# B&R Automation Studio project Nitto (part 17)

#### ac_loadRecipeMain.st
```iecst
(********************************************************************
 * COPYRIGHT -- Microsoft
 ********************************************************************
 * Programm: MAIN
 * Datei: ac_loadRecipeMain.st
 * Autor: awalz
 * Erstellt: 29. Juli 2014
 ********************************************************************
 * Implementierung des Programms MAIN
 ********************************************************************)

(* Fügt eine neue Aktion zum IEC Programm oder Bibliothek *)
ACTION ac_loadRecipeMain:

		// cutting units
		memcpy(ADR(machine.cuttingunit1.data.recipe),ADR(gApplRecipe.cutUnit1),SIZEOF(machine.cuttingunit1.data.recipe));
		memcpy(ADR(machine.cuttingunit2.data.recipe),ADR(gApplRecipe.cutUnit2),SIZEOF(machine.cuttingunit2.data.recipe));
		memcpy(ADR(machine.cuttingunit1.data.general),ADR(gApplRecipe.general),SIZEOF(machine.cuttingunit1.data.general));
		memcpy(ADR(machine.cuttingunit2.data.general),ADR(gApplRecipe.general),SIZEOF(machine.cuttingunit2.data.general));
		memcpy(ADR(machine.cuttingunit1.data.machdata),ADR(gMachRecipe.cut1),SIZEOF(machine.cuttingunit1.data.machdata));
		memcpy(ADR(machine.cuttingunit2.data.machdata),ADR(gMachRecipe.cut2),SIZEOF(machine.cuttingunit2.data.machdata));
//		machine.cuttingunit2.ctrl.getNextCuttPos.setCutOffset.UpdateRecipe := TRUE;
//		machine.cuttingunit2.ctrl.getNextCuttPos.setCutOffset.setvalueVisuRecipe := gApplRecipe.cutUnit2.RmOffset;
	(*	machine.cuttingunit1.data.machdata.position := 1000000;*)
		machine.cuttingunit1.data.general.periodLength := gApplRecipe.general.periodLength;
		machine.cuttingunit1.data.recipe.tool.gearRatioMotor := 5;(* weil die mit 0 überschrieben werden da der Krebs wieder Misst gebaut hat*)
		machine.cuttingunit1.data.recipe.tool.cogmodul :=3175.0;
		machine.cuttingunit1.data.newRecipe := TRUE;
		machine.cuttingunit2.data.recipe.tool.gearRatioMotor := 5;
		machine.cuttingunit2.data.recipe.tool.cogmodul :=3175.0;
	(*	machine.cuttingunit2.data.machdata.position := 3400000;*)
		machine.cuttingunit2.data.general.periodLength := gApplRecipe.general.periodLength;
		machine.cuttingunit2.markpoints.RegMarkPosition := -540000;
		machine.cuttingunit2.data.machdata.position := 850000;
		machine.cuttingunit2.data.newRecipe := TRUE;
//		machine.cuttingunit2.markpoints.RegMarkPosition := -540000; //Abstand vom Sensor zu Stanzmitte

		machine.masterModul.data.lenght1 := gApplRecipe.general.lenght1;
		machine.masterModul.data.lenght1 := gApplRecipe.general.lenght1;

		// master // general
		machine.masterModul.data.maxSpeed := gApplRecipe.general.maxVelocity;
		machine.masterModul.data.periodLength := gApplRecipe.general.periodLength;
		machine.masterModul.data.startSpeed := gApplRecipe.general.startVelocity;
		machine.masterModul.data.lenght1 := gApplRecipe.general.lenght1;
		machine.masterModul.data.lenght2 := gApplRecipe.general.lenght2;
		machine.masterModul.data.speedToCycleWebturrit := gApplRecipe.general.speedToCycleWebturrit;

		// unwinder drive side
		machine.UnwinderUnit.unwinderDrv.data.recipeData.maxDiamTension := gApplRecipe.UnwinderDrvSide.maxDiamTension;
		machine.UnwinderUnit.unwinderDrv.data.recipeData.minDiamTension := gApplRecipe.UnwinderDrvSide.minDiamTension;
		machine.UnwinderUnit.unwinderDrv.data.recipeData.mode := gApplRecipe.UnwinderDrvSide.mode;
		machine.UnwinderUnit.unwinderDrv.data.recipeData.reverse := gApplRecipe.UnwinderDrvSide.reverse;
		machine.UnwinderUnit.unwinderDrv.data.recipeData.warnDiam := gApplRecipe.UnwinderDrvSide.warnDiam;
		machine.UnwinderUnit.unwinderDrv.data.recipeData.stopDiam := gApplRecipe.UnwinderDrvSide.stopDiam;
		machine.UnwinderUnit.unwinderDrv.data.machData.axistyp := 1;	(*(-1: winder, +1: unwinder).*)
		// unwinder op side
		machine.UnwinderUnit.unwinderOp.data.recipeData.maxDiamTension := gApplRecipe.UnwinderOpSide.maxDiamTension;
		machine.UnwinderUnit.unwinderOp.data.recipeData.minDiamTension := gApplRecipe.UnwinderOpSide.minDiamTension;
		machine.UnwinderUnit.unwinderOp.data.recipeData.mode := gApplRecipe.UnwinderOpSide.mode;
		machine.UnwinderUnit.unwinderOp.data.recipeData.reverse := gApplRecipe.UnwinderOpSide.reverse;
		machine.UnwinderUnit.unwinderOp.data.recipeData.warnDiam := gApplRecipe.UnwinderOpSide.warnDiam;
		machine.UnwinderUnit.unwinderOp.data.recipeData.stopDiam := gApplRecipe.UnwinderOpSide.stopDiam;
		machine.UnwinderUnit.unwinderOp.data.machData.axistyp := 1;(*(-1: winder, +1: unwinder).*)
		// grid winder left
		machine.turngridwinder.gridwinderleft.data.recipeData.maxDiamTension := gApplRecipe.gridwinderleft.maxDiamTension;
		machine.turngridwinder.gridwinderleft.data.recipeData.minDiamTension := gApplRecipe.gridwinderleft.minDiamTension;
		machine.turngridwinder.gridwinderleft.data.recipeData.mode := gApplRecipe.gridwinderleft.mode;
		machine.turngridwinder.gridwinderleft.data.recipeData.reverse := gApplRecipe.gridwinderleft.reverse;
		machine.turngridwinder.gridwinderleft.data.recipeData.warnDiam := gApplRecipe.gridwinderleft.warnDiam;
		machine.turngridwinder.gridwinderleft.data.recipeData.stopDiam := gApplRecipe.gridwinderleft.stopDiam;
		machine.turngridwinder.gridwinderleft.data.machData.axistyp := - 1;(*(-1: winder, +1: unwinder).*)

		// grid winder right
		machine.turngridwinder.gridwinderright.data.recipeData.maxDiamTension := gApplRecipe.gridwinderright.maxDiamTension;
		machine.turngridwinder.gridwinderright.data.recipeData.minDiamTension := gApplRecipe.gridwinderright.minDiamTension;
		machine.turngridwinder.gridwinderright.data.recipeData.mode := gApplRecipe.gridwinderright.mode;
		machine.turngridwinder.gridwinderright.data.recipeData.reverse := gApplRecipe.gridwinderright.reverse;
		machine.turngridwinder.gridwinderright.data.recipeData.warnDiam := gApplRecipe.gridwinderright.warnDiam;
		machine.turngridwinder.gridwinderright.data.recipeData.stopDiam := gApplRecipe.gridwinderright.stopDiam;
		machine.turngridwinder.gridwinderright.data.machData.axistyp := - 1;
		// catch belt
		machine.catchbelt.ctrl.mode := gApplRecipe.catchbelt.mode;
		machine.catchbelt.axis.setGearRatio.enable := gApplRecipe.catchbelt.offsetOnOff;
		machine.catchbelt.axis.setGearRatio.UpdateRecipe := TRUE;
		machine.catchbelt.axis.setGearRatio.setvalueVisuRecipe := gApplRecipe.catchbelt.setvaluevisu;

		// conveyor
		machine.conveyor.ctrl.mode := gApplRecipe.conveyor.mode;
		machine.conveyor.axis.setGearRatio.enable := gApplRecipe.conveyor.offsetOnOff;
		machine.conveyor.axis.setGearRatio.UpdateRecipe := TRUE;
		machine.conveyor.axis.setGearRatio.setvalueVisuRecipe := gApplRecipe.conveyor.setvaluevisu;
		machine.conveyor.counters.setPieces := gApplRecipe.conveyor.setPieces;
		machine.conveyor.counters.validpieces := gApplRecipe.conveyor.validPieces;
		// long cuttter
		machine.longcutter.ctrl.mode := gApplRecipe.longcutter.mode;
		machine.longcutter.axis.setGearRatio.enable := gApplRecipe.longcutter.offsetOnOff;
		machine.longcutter.axis.setGearRatio.UpdateRecipe := TRUE;
		machine.longcutter.axis.setGearRatio.setvalueVisuRecipe := gApplRecipe.longcutter.setvaluevisu;

		// pull break station (pull belt)
		machine.pullbreakSt.axis.setGearRatio.enable := gApplRecipe.pullbelt.offsetOnOff;
		machine.pullbreakSt.axis.setGearRatio.UpdateRecipe := TRUE;
		machine.pullbreakSt.axis.setGearRatio.setvalueVisuRecipe := gApplRecipe.pullbelt.setvaluevisu;

		// Webbuffer
		machine.webbuffer.data.recipe.mode := gApplRecipe.tensionMeas.mode;
		machine.webbuffer.data.recipe.SetTension := gApplRecipe.tensionMeas.webTension;
END_ACTION
```

#### ac_loadMach_toRecipeMain.st
```iecst
(********************************************************************
 * COPYRIGHT -- Microsoft
 ********************************************************************
 * Programm: MAIN
 * Datei: ac_loadMach_toRecipeMain.st
 * Autor: awalz
 * Erstellt: 29. Juli 2014
 ********************************************************************
 * Implementierung des Programms MAIN
 ********************************************************************)

(* Fügt eine neue Aktion zum IEC Programm oder Bibliothek *)
ACTION ac_loadMach_toRecipeMain:

		// 2012-12-19 /schoenefeldr/
		// Copy recipe data from application recipe (actually active in the machine) into the selected recipe
		memcpy(ADR(RecipeEdit.cutUnit1),ADR(machine.cuttingunit1.data.recipe),SIZEOF(RecipeEdit.cutUnit1));
		memcpy(ADR(RecipeEdit.cutUnit2),ADR(machine.cuttingunit2.data.recipe),SIZEOF(RecipeEdit.cutUnit2));

//		RecipeEdit.cutUnit1.RmOffset := machine.cuttingunit1.ctrl.getNextCuttPos.setCutOffset.setvalueVisu;	 // OKrebs 15.09.14 //Damit der richtige Offsetwert in die perm Daten geschrieben wird
//		RecipeEdit.cutUnit2.RmOffset := machine.cuttingunit2.ctrl.getNextCuttPos.setCutOffset.setvalueVisu;  // OKrebs 15.09.14 //Damit der richtige Offsetwert in die perm Daten geschrieben wird
		RecipeEdit.general.lenght1 := machine.masterModul.data.lenght1; // OKrebs 17.09.14
		RecipeEdit.general.lenght2 := machine.masterModul.data.lenght2; // OKrebs 17.09.14
		RecipeEdit.general.speedToCycleWebturrit := machine.masterModul.data.speedToCycleWebturrit;

		machine.cuttingunit1.data.recipe.tool.gearRatioMotor := 5;(* weil die mit 0 überschrieben werden da der Krebs wieder Misst gebaut hat*)
		machine.cuttingunit1.data.recipe.tool.cogmodul :=3175.0;
		machine.cuttingunit2.data.recipe.tool.gearRatioMotor := 5;
		machine.cuttingunit2.data.recipe.tool.cogmodul :=3175.0;
		machine.cuttingunit2.markpoints.RegMarkPosition := -540000;
		machine.cuttingunit2.data.machdata.position := 850000;
		machine.cuttingunit2.data.general.periodLength := gApplRecipe.general.periodLength; //460000;
		(*machine.cuttingunit2.data.recipe.RmOffset*); (* muss noch irgendwie zu ende gebracht werden*)

		// unwinder drive side
		RecipeEdit.UnwinderDrvSide.maxDiamTension := machine.UnwinderUnit.unwinderDrv.data.recipeData.maxDiamTension;
		RecipeEdit.UnwinderDrvSide.minDiamTension := machine.UnwinderUnit.unwinderDrv.data.recipeData.minDiamTension;
		RecipeEdit.UnwinderDrvSide.mode := machine.UnwinderUnit.unwinderDrv.data.recipeData.mode;
		RecipeEdit.UnwinderDrvSide.reverse := machine.UnwinderUnit.unwinderDrv.data.recipeData.reverse;
		RecipeEdit.UnwinderDrvSide.warnDiam := machine.UnwinderUnit.unwinderDrv.data.recipeData.warnDiam;
		RecipeEdit.UnwinderDrvSide.stopDiam := machine.UnwinderUnit.unwinderDrv.data.recipeData.stopDiam;
//		RecipeEdit.UnwinderDrvSide.data.machData.GEAR_RATIO := 8;(*gMachRecipe.UnwinderDrvSide.GEAR_RATIO;*)
//		RecipeEdit.UnwinderDrvSide.machData.axistyp := 1;	(*(-1: winder, +1: unwinder).*)
		// unwinder op side
		RecipeEdit.UnwinderOpSide.maxDiamTension := machine.UnwinderUnit.unwinderOp.data.recipeData.maxDiamTension;
		RecipeEdit.UnwinderOpSide.minDiamTension := machine.UnwinderUnit.unwinderOp.data.recipeData.minDiamTension;
		RecipeEdit.UnwinderOpSide.mode := machine.UnwinderUnit.unwinderOp.data.recipeData.mode;
		RecipeEdit.UnwinderOpSide.reverse := machine.UnwinderUnit.unwinderOp.data.recipeData.reverse;
		RecipeEdit.UnwinderOpSide.warnDiam := machine.UnwinderUnit.unwinderOp.data.recipeData.warnDiam;
		RecipeEdit.UnwinderOpSide.stopDiam := machine.UnwinderUnit.unwinderOp.data.recipeData.stopDiam;
//		RecipeEdit.unwinderOp.data.machData.GEAR_RATIO := 8; (*gMachRecipe.UnwinderOpSide.GEAR_RATIO;*)
//		RecipeEdit.unwinderOp.data.machData.axistyp := 1;(*(-1: winder, +1: unwinder).*)
		// grid winder left
		RecipeEdit.gridwinderleft.maxDiamTension := machine.turngridwinder.gridwinderleft.data.recipeData.maxDiamTension;
		RecipeEdit.gridwinderleft.minDiamTension := machine.turngridwinder.gridwinderleft.data.recipeData.minDiamTension;
		RecipeEdit.gridwinderleft.mode := machine.turngridwinder.gridwinderleft.data.recipeData.mode;
		RecipeEdit.gridwinderleft.reverse := machine.turngridwinder.gridwinderleft.data.recipeData.reverse;
		RecipeEdit.gridwinderleft.warnDiam := machine.turngridwinder.gridwinderleft.data.recipeData.warnDiam;
		RecipeEdit.gridwinderleft.stopDiam := machine.turngridwinder.gridwinderleft.data.recipeData.stopDiam;
//		RecipeEdit.gridwinderleft.data.machData.GEAR_RATIO := 3; (*gMachRecipe.gridwinderleft.GEAR_RATIO;*)
//		RecipeEdit.gridwinderleft.data.machData.axistyp := - 1;(*(-1: winder, +1: unwinder).*)
		// grid winder right
		RecipeEdit.gridwinderright.maxDiamTension := machine.turngridwinder.gridwinderright.data.recipeData.maxDiamTension;
		RecipeEdit.gridwinderright.minDiamTension := machine.turngridwinder.gridwinderright.data.recipeData.minDiamTension;
		RecipeEdit.gridwinderright.mode := machine.turngridwinder.gridwinderright.data.recipeData.mode;
		RecipeEdit.gridwinderright.reverse := machine.turngridwinder.gridwinderright.data.recipeData.reverse;
		RecipeEdit.gridwinderright.warnDiam := machine.turngridwinder.gridwinderright.data.recipeData.warnDiam;
		RecipeEdit.gridwinderright.stopDiam := machine.turngridwinder.gridwinderright.data.recipeData.stopDiam;
//		RecipeEdit.gridwinderright.data.machData.GEAR_RATIO := 3; (*gMachRecipe.gridwinderleft.GEAR_RATIO;*)
//		RecipeEdit.gridwinderright.data.machData.axistyp := - 1;(*(-1: winder, +1: unwinder).*)
		// catch belt
		RecipeEdit.catchbelt.mode := machine.catchbelt.ctrl.mode;
		RecipeEdit.catchbelt.offsetOnOff := machine.catchbelt.axis.setGearRatio.enable;
		RecipeEdit.catchbelt.setvaluevisu := machine.catchbelt.axis.setGearRatio.setvalueVisu;

		// conveyor
		RecipeEdit.conveyor.mode := machine.conveyor.ctrl.mode;
		RecipeEdit.conveyor.offsetOnOff := machine.conveyor.axis.setGearRatio.enable;
		RecipeEdit.conveyor.setvaluevisu := machine.conveyor.axis.setGearRatio.setvalueVisu;

		// long cuttter
		RecipeEdit.longcutter.mode := machine.longcutter.ctrl.mode;
		RecipeEdit.longcutter.offsetOnOff := machine.longcutter.axis.setGearRatio.enable;
		RecipeEdit.longcutter.setvaluevisu := machine.longcutter.axis.setGearRatio.setvalueVisu;

		// pull break station (pull belt)
		RecipeEdit.pullbelt.offsetOnOff := machine.pullbreakSt.axis.setGearRatio.enable;
		RecipeEdit.pullbelt.setvaluevisu := machine.pullbreakSt.axis.setGearRatio.setvalueVisu;

		// Webbuffer Tension
		RecipeEdit.tensionMeas.mode := machine.webbuffer.data.recipe.mode;
		RecipeEdit.tensionMeas.webTension := machine.webbuffer.data.recipe.SetTension;
		/////////////////////////////////////////////////////////////////////////////////////////////////////////////////////////////

END_ACTION
```

#### ac_saveMachData.st
```iecst
(********************************************************************
 * COPYRIGHT -- Microsoft
 ********************************************************************
 * Programm: MAIN
 * Datei: ac_saveMachData.st
 * Autor: okrebs
 * Erstellt: 30. Juli 2014
 ********************************************************************
 * Implementierung des Programms MAIN
 ********************************************************************)

(* speichern der Maschinendaten zu MAIN_Variablen *)
ACTION ac_saveMachData:

		// distances
		machine.cuttingunit2.data.machdata.position := 850000;
		machine.cuttingunit1.data.recipe.tool.gearRatioMotor := 5;(* weil die mit 0 überschrieben werden da der Krebs wieder Misst gebaut hat*)
		machine.cuttingunit1.data.recipe.tool.cogmodul :=3175.0;
		machine.cuttingunit2.data.recipe.tool.gearRatioMotor := 5;
		machine.cuttingunit2.data.recipe.tool.cogmodul :=3175.0;
		machine.cuttingunit2.markpoints.RegMarkPosition := -540000;
	(*	machine.cuttingunit2.data.machdata.position := 540000;*)

		// unwinder drive side
		machine.UnwinderUnit.unwinderDrv.data.machData.coreDiam := gMachRecipe.UnwinderDrvSide.coreDiam;
		machine.UnwinderUnit.unwinderDrv.data.machData.frictionCompensation := gMachRecipe.UnwinderDrvSide.frictionCompensation;
		machine.UnwinderUnit.unwinderDrv.data.machData.GEAR_RATIO := 8;(*gMachRecipe.UnwinderDrvSide.GEAR_RATIO;*)
		machine.UnwinderUnit.unwinderDrv.data.machData.velocityOverride := gMachRecipe.UnwinderDrvSide.velocityOverride;
		machine.UnwinderUnit.unwinderDrv.data.machData.axistyp := 1;	(*(-1: winder, +1: unwinder).*)
		// unwinder op side
		machine.UnwinderUnit.unwinderOp.data.machData.coreDiam := gMachRecipe.UnwinderOpSide.coreDiam;
		machine.UnwinderUnit.unwinderOp.data.machData.frictionCompensation := gMachRecipe.UnwinderOpSide.frictionCompensation;
		machine.UnwinderUnit.unwinderOp.data.machData.GEAR_RATIO := 8; (*gMachRecipe.UnwinderOpSide.GEAR_RATIO;*)
		machine.UnwinderUnit.unwinderOp.data.machData.velocityOverride := gMachRecipe.UnwinderOpSide.velocityOverride;
		machine.UnwinderUnit.unwinderOp.data.machData.axistyp := 1;(*(-1: winder, +1: unwinder).*)
		// grid winder left
		machine.turngridwinder.gridwinderleft.data.machData.coreDiam := gMachRecipe.gridwinderleft.coreDiam;
		machine.turngridwinder.gridwinderleft.data.machData.frictionCompensation := gMachRecipe.gridwinderleft.frictionCompensation;
		machine.turngridwinder.gridwinderleft.data.machData.GEAR_RATIO := 3; (*gMachRecipe.gridwinderleft.GEAR_RATIO;*)
		machine.turngridwinder.gridwinderleft.data.machData.velocityOverride := gMachRecipe.gridwinderleft.velocityOverride;
		machine.turngridwinder.gridwinderleft.data.machData.axistyp := - 1;(*(-1: winder, +1: unwinder).*)
		// grid winder right
		machine.turngridwinder.gridwinderright.data.machData.coreDiam := gMachRecipe.gridwinderright.coreDiam;
		machine.turngridwinder.gridwinderright.data.machData.frictionCompensation := gMachRecipe.gridwinderright.frictionCompensation;
		machine.turngridwinder.gridwinderright.data.machData.GEAR_RATIO := 3; (*gMachRecipe.gridwinderright.GEAR_RATIO;*)
		machine.turngridwinder.gridwinderright.data.machData.velocityOverride := gMachRecipe.gridwinderright.velocityOverride;
		machine.turngridwinder.gridwinderright.data.machData.axistyp := - 1;
		// pack belt
		machine.packbelt.data.acceleration	:= gMachRecipe.botTandemWind.WarnDiam;
		machine.packbelt.data.deceleration	:= gMachRecipe.botTandemWind.StopDiam;
		machine.packbelt.data.highSpeed		:= gMachRecipe.botTandemWind.MaxPressure;
		machine.packbelt.data.lowSpeed		:= gMachRecipe.botTandemWind.MinPressure;

END_ACTION
```

### Program Logical/MainMachineCtrl/dummy (IEC) - Programm

#### dummyCyclic.st - Zyklischer Code
```iecst
(********************************************************************
 * COPYRIGHT -- Microsoft
 ********************************************************************
 * Programm: dummy
 * Datei: dummyCyclic.st
 * Autor: awalz
 * Erstellt: 26. Juni 2014
 ********************************************************************
 * Implementierung des Programms dummy
 ********************************************************************)

PROGRAM _CYCLIC

(* TODO : Code hier einfügen *)

END_PROGRAM
```

#### dummyInit.st - Initialisierungscode
```iecst
(********************************************************************
 * COPYRIGHT -- Microsoft
 ********************************************************************
 * Programm: dummy
 * Datei: dummyInit.st
 * Autor: awalz
 * Erstellt: 26. Juni 2014
 ********************************************************************
 * Implementierung des Programms dummy
 ********************************************************************)

PROGRAM _INIT

(* TODO : Code hier einfügen *)
	gUnwinder := gUnwinder;
	gMaster1 := gMaster1; (*Virtueller Master*)
	gCut1 := gCut1; (*Stanzstation 1*)
	gCut2 := gCut2; (*Stanzstation 2*)
	gGridLeft := gGridLeft; (*Gitteraufwickler 1*)
	gGridRight := gGridRight; (*Gitteraufwickler 2*)
	gPBS1 := gPBS1; (*Zugstation 1*)
	gPBS2 := gPBS2; (*Zugstation 1*)
	gCatchBelt := gCatchBelt; (*Fangband*)
	gConvBelt := gConvBelt; (*Auslageband*)
	gUnwOp := gUnwOp; (*Abwickler Operatorseite*)
	gUnwDrv := gUnwDrv; (*Abwickler Antriebsseite*)
	gBuffer := gBuffer; (*Bahnspeicher*)
	gGridFeeder := gGridFeeder; (*Drehvorrichtung Gitterturm*)
	gLongCut := gLongCut; (*Drehvorrichtung Gitterturm*)
	gUnwFeeder := gUnwFeeder;
	gUnwFeeder_HW := gUnwFeeder_HW;
	gUnwFeeder_DrvIf := gUnwFeeder_DrvIf;
	gUnwFeeder_DiDoIf := gUnwFeeder_DiDoIf;
	gUnwFeeder_ModuleOk := gUnwFeeder_ModuleOk;
	// neu // OKrebs // 23.11.16
	gPackBelt := gPackBelt;
	gPackBelt_HW := gPackBelt_HW;
	gPackBelt_DrvIf := gPackBelt_DrvIf;
	gPackBelt_DiDoIf := gPackBelt_DiDoIf;
	gPackBelt_ModuleOk := gPackBelt_ModuleOk;
	// ende neu
END_PROGRAM
```

- Visualisation Logical/Visualization (not shown)

### Package Logical/pkgRecipe - recipe handling

### Program Logical/pkgRecipe/save2USB (IEC) - copy recipes from CF to USB

#### save2USB.st - Implementation code
```iecst
(********************************************************************
 * COPYRIGHT -- Bernecker + Rainer
 ********************************************************************
 * Program: USB_Test
 * File: USB_Test.st
 * Author: beutert
 * Created: February 10, 2012
 ********************************************************************
 * Implementation of program USB_Test
 ********************************************************************)

PROGRAM _INIT

LayerMessageBoxErrorUSB := INVISIBLE;
LayerMessageBoxCopyOkUSB := INVISIBLE;
strcpy(ADR(szRecipeDirName), ADR('Recipes'));
strcpy(ADR(szToolDirName), ADR('Tools'));

strcpy(ADR(szDirName), ADR(szRecipeDirName));

END_PROGRAM

PROGRAM _CYCLIC

IF (BackupRecipes2USB = TRUE) THEN
	BackupRecipes2USB := FALSE;
	strcpy(ADR(szDirName), ADR(szRecipeDirName));
	StartBackup2USB := TRUE;
END_IF;
IF (BackupTools2USB = TRUE) THEN
	BackupTools2USB := FALSE;
	strcpy(ADR(szDirName), ADR(szToolDirName));
	StartBackup2USB := TRUE;
END_IF;

CASE bStep OF
	ST_WAIT:
		IF (StartBackup2USB = TRUE) THEN
			bStep := CREATE_NODE_ID_LIST;
		END_IF;

	CREATE_NODE_ID_LIST:
		bStepOld := bStep;
		UsbNodeListGet_0.enable 									:= 1;
		UsbNodeListGet_0.pBuffer 									:= ADR(lNodeIdBuffer);
		UsbNodeListGet_0.bufferSize 							:= SIZEOF(lNodeIdBuffer);
		UsbNodeListGet_0.filterInterfaceClass 		:= asusb_CLASS_MASS_STORAGE;  (*set filter on mass storage devices*)
		UsbNodeListGet_0.filterInterfaceSubClass 	:= 0;	(*no filter is set *)
		UsbNodeListGet_0();

		wStatus := UsbNodeListGet_0.status;
		IF (wStatus = 0) THEN
    	bStep := READ_DEVICE_DATA;
		ELSIF UsbNodeListGet_0.status = ERR_FUB_BUSY THEN
			(* call FUB again *)
		ELSE
			bStep := ERROR_STEP;
		END_IF;

	READ_DEVICE_DATA:
		bStepOld := bStep;
		UsbNodeGet_0.enable 		:= 1;
		UsbNodeGet_0.nodeId 		:= lNodeIdBuffer[bNode];  				(*specific node is read out of node_id_buffer*)
		UsbNodeGet_0.pBuffer 		:= ADR(UsbDataBuffer[bNode]);  		(*data of specific node get stored in usb_data_buffer*)
		UsbNodeGet_0.bufferSize := SIZEOF(UsbDataBuffer[bNode]);  (*size of specific node is read out usb_data_buffer*)
		UsbNodeGet_0();

		wStatus := UsbNodeGet_0.status;

		IF (wStatus = 0) THEN
			bNode := bNode + 1;  (*next node to be read out of buffer*)
			IF (bNode = UsbNodeListGet_0.listNodes) THEN  (*last existing node is reached*)
				bNode := 0;
				bStep := GET_DESCRIPTOR;  (*all nodes are read out of buffer*)
			END_IF;
		ELSIF (wStatus = ERR_FUB_BUSY) THEN
			(* call FUB again *)
		ELSE
			bStep := ERROR_STEP;
		END_IF;

	GET_DESCRIPTOR:
		bStepOld := bStep;
		UsbDescriptorGet_0.enable 				:= 1;
		UsbDescriptorGet_0.nodeId 				:= lNodeIdBuffer[bNode];  (*specific node is read out of node_id_buffer*)
		UsbDescriptorGet_0.requestType 		:= 0;  (*Request for device*)
    UsbDescriptorGet_0.descriptorType := 1;  (*Determines the device descriptor*)
		UsbDescriptorGet_0.languageId 		:= 0;  (*for device and configuration descriptors*)
		UsbDescriptorGet_0.pBuffer 				:= ADR(DeviceDescriptor[bNode]);  (*descriptor-data of specific node get stored in device_descriptor-buffer*)
		UsbDescriptorGet_0.bufferSize 		:= SIZEOF(DeviceDescriptor[bNode]);  (*size of specific node is read out device_descriptor-buffer*)
		UsbDescriptorGet_0();

		wStatus := UsbDescriptorGet_0.status;

		IF (wStatus = 0) THEN
			bNode := bNode + 1;  (*next node to be read out of buffer*)
			IF (bNode = UsbNodeListGet_0.listNodes) THEN  (*last existing node is reached*)
				bNode := 0;
				bStep := CREATE_FILE_DEVICE;  (*all nodes are read out of buffer*)
			END_IF;
		ELSIF (wStatus = ERR_FUB_BUSY) THEN
			(* call FUB again *)
		ELSE
			bStep := ERROR_STEP;
		END_IF;

	CREATE_FILE_DEVICE:
		bStepOld := bStep;
		strcpy(ADR(szDeviceName), ADR('USBSTICK'));  (*fixed Device-Name get copied to device_name-Variable*)

		strcpy(ADR(szDeviceParam), ADR('/DEVICE='));  (*first part of parameter get copied to device_param-Variable*)
		strcat(ADR(szDeviceParam), ADR(UsbDataBuffer[0].ifName));  (*second part get added to device_param-Variable*)

		DevLink_0.enable  := 1;
		DevLink_0.pDevice := ADR(szDeviceName);  (*Devicename is assigned*)
		DevLink_0.pParam  := ADR(szDeviceParam);  (*the path of the Device is assigned*)
		DevLink_0();

		wStatus := DevLink_0.status;

		IF (wStatus = 0) THEN
			xDevLinkDone := TRUE;
			bStep := DIRECTORY_INFO;
		ELSIF (wStatus = ERR_FUB_BUSY) THEN
			(* call FUB again *)
		ELSE
			bStep := ERROR_STEP;
		END_IF;

	DIRECTORY_INFO:
		bStepOld := bStep;
		DirInfo_0.enable 	:= 1;
		DirInfo_0.pDevice := ADR(szDeviceName);
		DirInfo_0.pPath 	:= ADR(szDirName);	// ADR('Recipes');
		DirInfo_0();

		wStatus := DirInfo_0.status;

		IF (wStatus = 0) THEN
			bStep := DIRECTORY_COPY;
		ELSIF (wStatus = ERR_FUB_BUSY) THEN
			(* call FUB again *)
		ELSIF  (wStatus = fiERR_DIR_NOT_EXIST) THEN
			bStep := DIRECTORY_CREATE;
		ELSE
			bStep := ERROR_STEP;
		END_IF;

	DIRECTORY_CREATE:
		bStepOld := bStep;
		DirCreate_0.enable 	:= 1;
		DirCreate_0.pDevice := ADR(szDeviceName);
		DirCreate_0.pName 	:= ADR(szDirName);	//ADR('Recipes');
		DirCreate_0();

		wStatus := DirCreate_0.status;

		IF (wStatus = 0) THEN
			bStep := DIRECTORY_COPY;
		ELSIF (wStatus = ERR_FUB_BUSY) THEN
			(* call FUB again *)
		ELSE
			bStep := ERROR_STEP;
		END_IF;

	DIRECTORY_COPY:
		DirCopy_0.enable 		:= 1;
		DirCopy_0.pSrcDev 	:= ADR('USERPART');
		DirCopy_0.pSrcDir 	:= ADR(szDirName);	//ADR('Recipes');;
		DirCopy_0.pDestDev 	:= ADR(szDeviceName);
		DirCopy_0.pDestDir 	:= ADR(szDirName);	//ADR('Recipes');
		DirCopy_0.option 		:= fiOVERWRITE;
		DirCopy_0();

		wStatus := DirCopy_0.status;

		IF (wStatus = 0) THEN
			bStep := UNLINK_DEVICE;
		ELSIF (wStatus = ERR_FUB_BUSY) THEN
			(* call FUB again *)
		ELSE
			bStep := ERROR_STEP;
		END_IF;

	UNLINK_DEVICE:
		bStepOld := bStep;
		DevUnlink_0.enable := 1;
		DevUnlink_0.handle := DevLink_0.handle;  (*handle from DevLink is assigned to cut the connection to specific file-device*)
		DevUnlink_0();

		wStatus := DevUnlink_0.status;

		IF (wStatus = 0) THEN
			xDevLinkDone := FALSE;
			bStep := FINISH;
		ELSIF (wStatus = ERR_FUB_BUSY) THEN
			(* call FUB again *)
		ELSE
			bStep := ERROR_STEP;
		END_IF;

	FINISH:  (*successfully finished*)
		bStepOld := bStep;
		StartBackup2USB := FALSE;
		LayerMessageBoxCopyOkUSB := VISIBLE;
		bStep := ST_WAIT;  (*back to beginning - wait for start_reading_usb_data to be set*)

	ERROR_STEP:	(*tbd: error-handling*)
		StartBackup2USB := FALSE;
		IF (xDevLinkDone = TRUE) THEN
			bStep := UNLINK_DEVICE;
		ELSE
			LayerMessageBoxErrorUSB := VISIBLE;
			bStep := ST_WAIT;  (*back to beginning - wait for start_reading_usb_data to be set*)
		END_IF;

END_CASE;

END_PROGRAM
```

#### save2USB.var - Local variables
```iecst
(********************************************************************
 * COPYRIGHT -- Bernecker + Rainer
 ********************************************************************
 * Program: USB_Test
 * File: USB_Test.var
 * Author: beutert
 * Created: February 10, 2012
 ********************************************************************
 * Local variables of program USB_Test
 ********************************************************************)
VAR
	szDeviceParam : STRING[80];
	UsbDescriptorGet_0 : UsbDescriptorGet;
	UsbDataBuffer : ARRAY[0..4] OF usbNode_typ;
	UsbNodeListGet_0 : UsbNodeListGet;
	bStep : USINT;
	szDeviceName : STRING[80];
	lNodeIdBuffer : ARRAY[0..4] OF UDINT;
	bStepOld : USINT;
	bNode : USINT;
	UsbNodeGet_0 : UsbNodeGet;
	DevLink_0 : DevLink;
	DeviceDescriptor : ARRAY[0..4] OF usbDeviceDescr_typ;
	DevUnlink_0 : DevUnlink;
	wStatus : UINT;
	StartBackup2USB : BOOL;
	BackupRecipes2USB : BOOL;
	BackupTools2USB : BOOL;
	DirInfo_0 : DirInfo;
	DirCopy_0 : DirCopy;
	DirCreate_0 : DirCreate;
END_VAR
VAR CONSTANT
	ST_WAIT : USINT := 0;
	CREATE_NODE_ID_LIST : USINT := 5;
	READ_DEVICE_DATA : USINT := 10;
	GET_DESCRIPTOR : USINT := 15;
	CREATE_FILE_DEVICE : USINT := 20;
	DIRECTORY_INFO : USINT := 25;
	DIRECTORY_CREATE : USINT := 30;
	DIRECTORY_COPY : USINT := 35;
	UNLINK_DEVICE : USINT := 45;
	FINISH : USINT := 250;
	ERROR_STEP : USINT := 255;
END_VAR
VAR
	xDevLinkDone : BOOL;
	LayerMessageBoxErrorUSB : USINT;
END_VAR
VAR CONSTANT
	INVISIBLE : USINT := 1;
	VISIBLE : USINT := 0;
END_VAR
VAR
	LayerMessageBoxCopyOkUSB : USINT;
	szRecipeDirName : STRING[80];
	szToolDirName : STRING[80];
	szDirName : STRING[80];
END_VAR
```

### Program Logical/pkgRecipe/csv_hdl (IEC) - file handling

#### csv_hdl.st - Implementation code
```iecst
(********************************************************************
 * COPYRIGHT -- Bernecker + Rainer
 ********************************************************************
 * Program: csv_hdl
 * File: csv_hdl.st
 * Author: beutert
 * Created: August 28, 2012
 ********************************************************************
 * Implementation of program csv_hdl
 ********************************************************************)

PROGRAM _INIT

	REPEAT
		VCHandle	:= VA_Setup(TRUE, 'Visu');
	UNTIL (VCHandle <> 0) END_REPEAT;

	CSV_Hndl.LayerMessageBoxOverwrite := INVISIBLE;
	CSV_Hndl.LayerMessageBoxDeleteFile := INVISIBLE;
	CSV_Hndl.LayerNewFileName := INVISIBLE;
	CSV_Hndl.LayerMessageBoxSaveFile := INVISIBLE;

	HWInfo_0.enable := TRUE;
	HWInfo_0.first := TRUE;
	HWInfo_0.pName := ADR(HWString);
	HWInfo_0();

	DirCreate_0.pDevice	:= ADR('USERPART');
	DirCreate_0.pName	:= ADR('Recipes');
	DirCreate_0.enable	:= TRUE;
	REPEAT
		DirCreate_0();
	UNTIL (DirCreate_0.status <> ERR_FUB_BUSY) END_REPEAT;

//	strcpy(ADR(szFileDevice), "USBSTICK");
//	strcpy(ADR(szFileDevice), "FLASH");
	strcpy(ADR(szFileDevice), ADR('DIR_RCP'));
	IF HWString = 'AR000' THEN
		strcpy(ADR(szDevLinkPara), ADR('/DEVICE=C:\\temp\\Recipes'));
		// 2012-12-13 /schoenefeldr/
		// In simulations mode: Always on highest password level
		Level_Passwort := 10;
	ELSE
		strcpy(ADR(szDevLinkPara), ADR('/DEVICE=F:\\Recipes'));
	END_IF

	DevLink_0.enable 	:= 1;
	DevLink_0.pDevice := ADR(szFileDevice);
	DevLink_0.pParam 	:= ADR(szDevLinkPara);
	DevLink_0();

	strcpy(ADR(CSV_Header.CustomerName),ADR('Spilker'));
	strcpy(ADR(CSV_Header.MachineNumber),ADR('Herpa Print'));
	strcpy(ADR(CSV_Header.SW_Version),ADR('Version V1.00'));

	//strcpy(ADR(RecipeEdit.MachineString),ADR('machine1'));

	pNames[0] :=  ADR('csv_hdl:tmpRecipe');		//Name der zu sichernden PV
//	pNames[1] :=  ADR('CSV_SearchData');				//mehrere möglich

	StructSizes[0] := SIZEOF(tmpRecipe);				//Größe der zu sichernden PV
//	StructSizes[1] := SIZEOF(CSV_SearchData);

	CSV_InitVariable.pStructName := ADR(pNames);
	CSV_InitVariable.NumOfStructs := 1;					//Anzahl der zu sichernden Elemente, wenn CSV_SearchData auch gesichert werden soll, muss hier 2 stehen
	CSV_InitVariable.FullNameLenght := 0;
	CSV_InitVariable.Options := 0;
	CSV_InitVariable();

  IF (CSV_InitVariable.status > 0) AND (CSV_InitVariable.status < ERR_FUB_BUSY) THEN
  	Step := ST_ERROR;
  ELSE
   	Step := ST_COMMAND;
	END_IF;

//Speicherplatz allokieren
	CSVInitCheckFileVersion.enable := 1;
	CSVInitCheckFileVersion.MemCounter := CSV_InitVariable.MemCounter;
	CSVInitCheckFileVersion();

  IF (CSVInitCheckFileVersion.status < 65535) AND (CSVInitCheckFileVersion.status > 0) THEN
    Step := ST_ERROR;
  ELSE
   	Step := ST_COMMAND;
		CSVInitCheckFileVersion.enable := 1;
		CSVInitCheckFileVersion.MemCounter := CSV_InitVariable.MemCounter;
		CSVInitCheckFileVersion();
	END_IF;

  IF (CSVInitCheckFileVersion.status < ERR_FUB_BUSY) AND (CSVInitCheckFileVersion.status > 0) THEN
    Step := ST_ERROR;
  ELSE
    Step := ST_COMMAND;
		CSV_Hndl.ReqDirRead := TRUE;
		xSorted := TRUE;
		OldListBoxIdx := 16#FFFF;
	END_IF;

END_PROGRAM

PROGRAM _CYCLIC

	IF Layer_Password THEN
		Show_Layer_password := 0;

		IF InputPassword =('1234') THEN
			Level_Passwort := 10;
		ELSE
				Level_Passwort := 0;
		END_IF;
	ELSE
		Show_Layer_password := 1;
		InputPassword :='****';
//		reset Passwort über Timer fehlt noch
//		Level_Passwort := 0 ;
	END_IF;

CASE Step OF

	(****************************************/
	/* command interface                    */
	/****************************************)
		ST_COMMAND:	(*0*)
			IF (CSV_Hndl.ReqDirRead) THEN
				IF (xSorted = TRUE) THEN
				Step := ST_LIST_FILE_SORT;
			ELSE
				Step := ST_LIST_FILE;
			END_IF;

		ELSIF (CSV_Hndl.ReqDelRecipe) THEN
			CSV_Hndl.ReqDelRecipe := FALSE;
			strcpy(ADR(CSV_Hndl.FileNameDelete),ADR(CSV_Hndl.ListboxFileNames[CSV_Hndl.ListboxIdx]));
			strcat(ADR(CSV_Hndl.FileNameDelete),ADR('.csv'));
			CSV_Hndl.LayerMessageBoxDeleteFile := VISIBLE;	//Message einblenden
		  CSV_Hndl.FileDelete := 0;
			Step := ST_ASK_FOR_DELETE_FILE;

		ELSIF (CSV_Hndl.ReqCreateNew) THEN
			CSV_Hndl.ReqCreateNew := FALSE;
//			memcpy(ADR(tmpRecipe), ADR(RecipeNew), SIZEOF(tmpRecipe));	//copy data structure
			Step := ST_SEARCH_DATA;

		ELSIF (CSV_Hndl.ReqParaWrite) THEN
			memcpy(ADR(tmpRecipe), ADR(RecipeEdit), SIZEOF(tmpRecipe)); 	//copy data structure global to local
			strcpy(ADR(CSV_Hndl.FileNameNew),ADR(CSV_Hndl.ListboxFileNames[CSV_Hndl.ListboxIdx]));
			strcat(ADR(CSV_Hndl.FileNameNew),ADR('.csv'));
			CSV_Hndl.OverwriteFile := TRUE;
			Step := ST_SEARCH_DATA;

		ELSIF (CSV_Hndl.ReqParaWriteAfterValueChanged) THEN
			CSV_Hndl.ReqParaWriteAfterValueChanged := FALSE;
			memcpy(ADR(tmpRecipe), ADR(tmpRecipeOld), SIZEOF(tmpRecipe)); 	//copy data structure
			strcpy(ADR(CSV_Hndl.FileNameNew),ADR(FileNameOld));
			strcat(ADR(CSV_Hndl.FileNameNew),ADR('.csv'));
			CSV_Hndl.OverwriteFile := TRUE;
			Step := ST_SEARCH_DATA;

		ELSIF (CSV_Hndl.ReqSaveRecipeAs) THEN
			CSV_Hndl.ReqSaveRecipeAs := FALSE;
			memcpy(ADR(tmpRecipe), ADR(RecipeEdit), SIZEOF(tmpRecipe));	//copy data structure
			Step := ST_SEARCH_DATA;

		ELSIF (CSV_Hndl.ReqParaRead) THEN
			Step := ST_READ_FILE;

//		ELSIF(Start_CheckVersion)THEN
//			Step:= ST_CHECK_VERSION;
		END_IF;

	(****************************************/
	/* list all CSV-files in a array-string */
	/****************************************)

	(*OHNE SORTIERUNG:*)
	(*csv-Dateien auf Device auflisten*)
	ST_LIST_FILE:	(*1*)
		StepOld := Step;
   	CSV_ListCSVFile.pStringArray := ADR(CSV_Hndl.ListboxFileNames[0]);
   	CSV_ListCSVFile.SizeStringArray := SIZEOF(CSV_Hndl.ListboxFileNames);
   	CSV_ListCSVFile.ArrayNum := SIZEOF(CSV_Hndl.ListboxFileNames) / SIZEOF(CSV_Hndl.ListboxFileNames[0]);
   	CSV_ListCSVFile.NumListboxLines := 10;
		CSV_ListCSVFile.pFileDevice := ADR(szFileDevice);
   	CSV_ListCSVFile.MaxNameLenght := 28;
   	CSV_ListCSVFile.command := FiJOB_CREATE_FILE_LIST; //2
   	CSV_ListCSVFile();

		IF (CSV_ListCSVFile.CSV_FileNum > 0) THEN
	    CSV_Hndl.ListboxMaxLines := CSV_ListCSVFile.CSV_FileNum  - 1;
	  ELSE
	  	CSV_Hndl.ListboxMaxLines := 0;
	  END_IF;

		//no error
	  IF (CSV_ListCSVFile.status = 0) THEN
			CSV_Hndl.ReqDirRead := 0;

			IF (CSV_Hndl.SetListBoxIdxToZero) THEN
				CSV_Hndl.SetListBoxIdxToZero := FALSE;
				CSV_Hndl.ListboxIdx := 0;
				CSV_Hndl.ListboxProgParaIdx := 0;
				CSV_Hndl.ReqParaRead := TRUE;
			END_IF;

	  	Step := ST_COMMAND;
		END_IF;

	   //error
	   IF ( (CSV_ListCSVFile.status <> 0) AND (CSV_ListCSVFile.status <> 65535) ) THEN
	      CSV_Hndl.ReqDirRead := 0;
	      Step := ST_ERROR;
	   END_IF;

	(*MIT SORTIERUNG:*)
	(*csv-Dateien auf Device auflisten*)
	ST_LIST_FILE_SORT:	(*2*)
		StepOld := Step;
   	CSV_ListCSVFile.pStringArray := ADR(FileNamesRead);
   	CSV_ListCSVFile.SizeStringArray := SIZEOF(FileNamesRead);
   	CSV_ListCSVFile.ArrayNum := SIZEOF(FileNamesRead) / SIZEOF(FileNamesRead[0]);
   	CSV_ListCSVFile.NumListboxLines := 10;
		CSV_ListCSVFile.pFileDevice := ADR(szFileDevice);
   	CSV_ListCSVFile.MaxNameLenght := 28;
   	CSV_ListCSVFile.command := 2;
   	CSV_ListCSVFile();

		IF (CSV_ListCSVFile.CSV_FileNum > 0) THEN
	    CSV_Hndl.ListboxMaxLines := CSV_ListCSVFile.CSV_FileNum  - 1;
	  ELSE
	  	CSV_Hndl.ListboxMaxLines := 0;
	  END_IF;

	  //no error
	  IF (CSV_ListCSVFile.status = 0) THEN
  		Step := ST_SORT_FILE_NAMES;
		END_IF;

	   //error
	   IF ( (CSV_ListCSVFile.status <> 0) AND (CSV_ListCSVFile.status <> 65535) ) THEN
	      CSV_Hndl.ReqDirRead := 0;
	      Step := ST_ERROR;
	   END_IF;

	(****************************************/
	/* sort FileNames                    */
	/****************************************)
	ST_SORT_FILE_NAMES:	(*9*)
		StepOld := Step;
    Sort_0.enable := TRUE;
		Sort_0.pStringArray := ADR(FileNamesRead);
		Sort_0.StringLen := SIZEOF(FileNamesRead[0]);
		Sort_0.ArrayLen := SIZEOF(FileNamesRead);
		Sort_0();

	  IF (Sort_0.Status = 0) THEN
	  	CSV_Hndl.ReqDirRead := 0;
			memcpy(ADR(CSV_Hndl.ListboxFileNames), ADR(FileNamesRead), SIZEOF(FileNamesRead));

			IF (CSV_Hndl.SetListBoxIdxToZero) THEN
				CSV_Hndl.SetListBoxIdxToZero := FALSE;
				CSV_Hndl.ListboxIdx := 0;
				CSV_Hndl.ListboxProgParaIdx := 0;
				CSV_Hndl.ReqParaRead := TRUE;
			END_IF;

	   	Step := ST_COMMAND;
	  END_IF;

	(*****************************************/
	/* search for the data from the variable */
	/*****************************************)
	ST_SEARCH_DATA:	(*3*)
		StepOld := Step;
//		memcpy(ADR(tmpRecipe), ADR(RecipeEdit), SIZEOF(tmpRecipe)); globale Datenstruktur auf lokale umkopieren
   	CSV_SearchData.pStructName := CSV_InitVariable.pStructName;
   	CSV_SearchData.NumOfStructs := CSV_InitVariable.NumOfStructs;
   	CSV_SearchData.pStructMem := CSV_InitVariable.pStructMem;
   	CSV_SearchData.MemLen := CSV_InitVariable.MemCounter;
   	CSV_SearchData.FullNameLenght := 0;
   	CSV_SearchData.Separator := 59;	//';';
   	CSV_SearchData.Options := 0;
   	CSV_SearchData.FileHeader := HEADER;
   	CSV_SearchData.pMaschineNo := ADR(CSV_Header.CustomerName);
   	CSV_SearchData.pComment := ADR(CSV_Header.MachineNumber);
   	CSV_SearchData.pVersion := ADR(CSV_Header.SW_Version);
   	CSV_SearchData();

   	//no error
   	IF (CSV_SearchData.status = 0) THEN
			strcpy(ADR(CSV_Hndl.FileNameSave), ADR(CSV_Hndl.FileNameNew));
			CSV_Hndl.ReqParaWrite := FALSE;
			Step := ST_REPLACE_WRONG_CHARS;
   	END_IF;

   	//error
	  IF ( (CSV_SearchData.status <> 0) AND (CSV_SearchData.status <> 65535) ) THEN
	  	Step := ST_ERROR;
		END_IF;

	(****************************************/
	/* Replace Wrong Signs                  */
	/****************************************)
	ST_REPLACE_WRONG_CHARS:	(*13*)
		StepOld := Step;
		IF (strlen(ADR(CSV_Hndl.FileNameSave)) <> 0) THEN
			//control, if the filename has the right extension
			strcpy(ADR(tmpString), ADR(''));

			FOR i:=0 TO strlen(ADR(CSV_Hndl.FileNameSave))-1 DO
				Dyn_Usint ACCESS (ADR(CSV_Hndl.FileNameSave) + i);
				strcpy(ADR(tmpChar), ADR(''));
				memcpy(ADR(tmpChar), ADR(CSV_Hndl.FileNameSave) + i, 1);
//				IF ( ((Dyn_Usint >= ADR('0') ) AND (Dyn_Usint <= ADR('9') )) OR
//				     ((Dyn_Usint >= ADR('A') ) AND (Dyn_Usint <= ADR('Z') )) OR
//						 ((Dyn_Usint >= ADR('a') ) AND (Dyn_Usint <= ADR('z') )) OR
//						 ( Dyn_Usint  = ADR('_') ) OR  (Dyn_Usint = ADR('-')   ) OR
//						 ( Dyn_Usint  = ADR('.') ) OR  (Dyn_Usint = 0) ) THEN
					IF (((Dyn_Usint >= 48) AND (Dyn_Usint <= 57)) OR
						  ((Dyn_Usint >= 65) AND (Dyn_Usint <= 90)) OR
						  ((Dyn_Usint >= 97) AND (Dyn_Usint <= 122)) OR
						   (Dyn_Usint  = 95) OR (Dyn_Usint = 45) OR
						   (Dyn_Usint  = 46) OR (Dyn_Usint = 0)) THEN
					//valid chars
					tmpString := CONCAT(tmpString, tmpChar);
				ELSE
					//non valid chars
					tmpString := CONCAT(tmpString, '-');
				END_IF;
			END_FOR;
		END_IF;	//(strlen(ADR(CSV_Hndl.FileNameSave)) <> 0)

		Step := ST_SEARCH_FILE_ON_USB;
		strcpy (ADR(CSV_Hndl.FileNameSave),ADR(tmpString));

	(****************************************/
	/* search filenames                    */
	/****************************************)
	ST_SEARCH_FILE_ON_USB:	(*12*)
		StepOld := Step;
	  CSV_SearchFile.pFileName := ADR(CSV_Hndl.FileNameSave);
		CSV_SearchFile.pDevice := ADR(szFileDevice);
 		CSV_SearchFile();

	  //no error No file Found
	  IF (CSV_SearchFile.status = 0) THEN
	  	Step := ST_WRITE_FILE;
		END_IF;
	  //no error File Found
	  IF (CSV_SearchFile.status = 1) THEN
			IF (CSV_Hndl.OverwriteFile) THEN
				CSV_Hndl.OverwriteFile := FALSE;
				Step := ST_WRITE_FILE;
			ELSE
				CSV_Hndl.LayerMessageBoxOverwrite := VISIBLE;	//Message einblenden
			  CSV_Hndl.FileOverWrite := 0;
		  	Step := ST_ASK_FOR_OVERWRITE_FILE;
			END_IF;
		END_IF;
	  //error
	  IF ((CSV_SearchFile.status > 1) AND (CSV_SearchFile.status <> ERR_FUB_BUSY)) THEN
	  	Step := ST_ERROR;
	  END_IF;

	(****************************************/
	/* ask for overwrite file               */
	/****************************************)
	ST_ASK_FOR_OVERWRITE_FILE:	(*11*)
		StepOld := Step;
		IF (CSV_Hndl.LayerMessageBoxOverwrite = INVISIBLE) THEN
			IF (CSV_Hndl.FileOverWrite = 0) THEN
				CSV_Hndl.ReqNewRecipe := 1;	//start dialogue again
				Step := ST_COMMAND;
			ELSE
   			Step := ST_WRITE_FILE;
				CSV_Hndl.FileOverWrite := 0;
	    END_IF;
		END_IF;

	(*****************************************/
	/* write the searched data in a CSV-file */
	/*****************************************)
	ST_WRITE_FILE:	(*4*)
		StepOld := Step;
	 	CSV_WriteCSVFile.pFileName := ADR(CSV_Hndl.FileNameSave);      ///  HIER !!!!!!
	  CSV_WriteCSVFile.pDevice := ADR(szFileDevice);
	 	CSV_WriteCSVFile.pStructMem := CSV_InitVariable.pStructMem;
	 	CSV_WriteCSVFile.MemLen := CSV_SearchData.FileLen;
	 	CSV_WriteCSVFile.Mode := FILE_OW;
	 	CSV_WriteCSVFile();

	  //no error
	  IF (CSV_WriteCSVFile.status = 0) THEN
	  	CSV_Hndl.ReqParaWrite := FALSE;
			CSV_Hndl.ReqDirRead := TRUE;		//read directory again after writing a (new) file
	    Step := ST_COMMAND;
	  END_IF;
	  //error
	  IF ((CSV_WriteCSVFile.status <> 0) AND (CSV_WriteCSVFile.status <> 65535)) THEN
			CSV_Hndl.ReqParaWrite := FALSE;
    	//Es sind nur Zeichen und Zahlen erlaubt
			IF (CSV_WriteCSVFile.status = 5004) THEN
				Step :=  ST_ERROR;
			END_IF;
			Step := ST_ERROR;
	 	END_IF;

	(*****************************************/
	/* read a CSV-file                       */
	/*****************************************)
	ST_READ_FILE:	(*5*)
		StepOld := Step;
	  CSV_ReadCSVFile.pFileName := ADR(CSV_Hndl.ListboxFileNames[CSV_Hndl.ListboxIdx]);
   	CSV_ReadCSVFile.pDevice := ADR(szFileDevice);
   	CSV_ReadCSVFile.No_DatatypControl := 1;
//   	CSV_ReadCSVFile.Options := 0;
   	CSV_ReadCSVFile.IgnoreError := 1;
   	CSV_ReadCSVFile.Separator := 59;	//';';
   	CSV_ReadCSVFile();

   	//no error
   	IF (CSV_ReadCSVFile.status = 0) THEN
     	CSV_Hndl.ReqParaRead := 0;
			memcpy(ADR(RecipeEdit), ADR(tmpRecipe), SIZEOF(RecipeEdit));
			CSV_Hndl.ListBoxRecipeChanged := 1;	//another recipe was selected
			SaveUserData := 1;
      Step := ST_COMMAND;
   	END_IF;

   	//error
   	IF ((CSV_ReadCSVFile.status <> 0) AND (CSV_ReadCSVFile.status <> 65535)) THEN
      CSV_Hndl.ReqParaRead := 0;
      Step := ST_ERROR;
	 END_IF;

	(*****************************************/
	/* read a CSV-file                       */
	/*****************************************)
	ST_CHECK_VERSION:	(*6*)
		StepOld := Step;
		CSVCheckFileVersion.enable := 1;
		CSVCheckFileVersion.pFileName := ADR('csv1.CSV');
		CSVCheckFileVersion.pDevice := ADR(szFileDevice);
		CSVCheckFileVersion.pStructSizes := ADR(StructSizes);
		CSVCheckFileVersion.NumOfStruct := CSV_InitVariable.NumOfStructs;
		CSVCheckFileVersion.pVersion := ADR('V0.02.2');
		CSVCheckFileVersion.pFileBuffer := CSVInitCheckFileVersion.pFileBuffer;
		CSVCheckFileVersion.FileBufferSize := CSVInitCheckFileVersion.FileBufferSize;
		CSVCheckFileVersion();

	  //no error
	 	IF (CSVCheckFileVersion.status = 0) THEN
	   	Step := ST_COMMAND;
	 	END_IF;

	  //error
	  IF ((CSVCheckFileVersion.status <> 0) AND (CSVCheckFileVersion.status <> 65535)) THEN
			Step := ST_ERROR;
   	END_IF;

	(****************************************/
	/* ask for delete file                  */
	/****************************************)
	ST_ASK_FOR_DELETE_FILE:	(*7*)
		StepOld := Step;
		IF (CSV_Hndl.LayerMessageBoxDeleteFile = INVISIBLE) THEN
			IF (CSV_Hndl.FileDelete = 0) THEN
				Step := ST_COMMAND;
			ELSE
				CSV_Hndl.FileDelete := 0;
   			Step := ST_DELETE_FILE;
	    END_IF;
		END_IF;

	(*****************************************/
	/* delete a CSV-file                       */
	/*****************************************)
	ST_DELETE_FILE:	(*8*)
		StepOld := Step;
		FileDelete_0.enable 	:= 1;
		FileDelete_0.pDevice 	:= ADR(szFileDevice);
		FileDelete_0.pName 		:= ADR(CSV_Hndl.FileNameDelete);
		FileDelete_0();

	  //no error
	 	IF (FileDelete_0.status = 0) THEN
			CSV_Hndl.ReqDirRead := TRUE;		//read directory again after deleting a file
			CSV_Hndl.SetListBoxIdxToZero := TRUE;
	   	Step := ST_COMMAND;
	 	END_IF;

	  //error
	  IF ((FileDelete_0.status <> 0) AND (FileDelete_0.status <> ERR_FUB_BUSY)) THEN
			Step := ST_ERROR;
   	END_IF;

	(****************************************/
	/* change the file device               */
	/****************************************)
	ST_UNLINK_DEVICE:	(*15*)
		StepOld := Step;
		DevUnlink_0.enable := 1;
		DevUnlink_0.handle := DevLink_0.handle;
		DevUnlink_0();

	  //no error
		IF (DevUnlink_0.status = 0) THEN
			Step := ST_LINK_DEVICE;
		ELSIF (DevUnlink_0.status = ERR_FUB_BUSY) THEN
			//
		ELSE
			Step := ST_ERROR;
		END_IF;

	ST_LINK_DEVICE:	(*16*)
		StepOld := Step;
		DevLink_0.enable 	:= 1;
		DevLink_0.pDevice := ADR(szFileDevice);
		DevLink_0.pParam 	:= ADR(szDevLinkPara);
		DevLink_0();

	  //no error
		IF (DevLink_0.status = 0) THEN
			CSV_Hndl.SetListBoxIdxToZero := TRUE;
			CSV_Hndl.ReqDirRead := TRUE;
			Step := ST_COMMAND;
		ELSIF (DevLink_0.status = ERR_FUB_BUSY) THEN
			//
		ELSE
			Step := ST_ERROR;
		END_IF;

	(****************************************/
	/* error counter                        */
	/****************************************)
	ST_ERROR:	(*255*)
	   Error := Error + 1;
	   Step := ST_COMMAND;

END_CASE;

(*************************************************************************
 ************************************************************************)
//copy the name of the selected csv file into a variable
IF ((CSV_Hndl.ListboxIdx >= 0) AND (CSV_Hndl.ListboxIdx < 100)) THEN
	strcpy(ADR(CSV_Hndl.FileNameSelected), ADR(CSV_Hndl.ListboxFileNames[CSV_Hndl.ListboxIdx]));
ELSE
	strcpy(ADR(CSV_Hndl.FileNameSelected),ADR('index out of range'));
END_IF;

//another recipe was selected in the list
IF (OldListBoxIdx <> CSV_Hndl.ListboxIdx) THEN
	IF (CSV_Hndl.ValueChanged) THEN			//a value was changed
		CSV_Hndl.ValueChanged := FALSE;
		memcpy(ADR(tmpRecipeOld), ADR(RecipeEdit), SIZEOF(tmpRecipeOld)); 	//copy data structure global to local
		strcpy(ADR(FileNameOld),  ADR(CSV_Hndl.ListboxFileNames[OldListBoxIdx]));
		CSV_Hndl.LayerMessageBoxSaveFile := VISIBLE;	//show messagebox
	END_IF;
	IF (CSV_Hndl.LayerMessageBoxSaveFile = INVISIBLE) THEN
		OldListBoxIdx := CSV_Hndl.ListboxIdx;
		CSV_Hndl.ReqParaRead := TRUE;

		CSV_Hndl.ListboxProgParaIdx := 0;	//set index of second listbox to 0
	END_IF;
END_IF;

//---------------------------------
//create a new recipe
IF(CSV_Hndl.BtnNew) THEN
	IF (CSV_Hndl.ReqNewRecipe = 1) THEN
		CSV_Hndl.ReqNewRecipe := 0;
		NewRecipe;	//call action: show layer and alpha pad
	END_IF;
	IF ((CSV_Hndl.NewFileNameEntered = TRUE) OR (CSV_Hndl.StatusNewFileName = 16384)) THEN
		CSV_Hndl.LayerNewFileName := INVISIBLE;
		//Name entered or escaped function ?
		IF (CSV_Hndl.NewFileNameEntered = TRUE) THEN
			//create structure with default values and write to file
			DefRecipe;																		   ///  HIER !!!!!!
			CSV_Hndl.ReqCreateNew := TRUE;
			CSV_Hndl.SetListBoxIdxToZero := TRUE;
		END_IF;

		CSV_Hndl.NewFileNameEntered := FALSE;
	END_IF;
END_IF;

//---------------------------------
//save a recipe under a new name
IF (CSV_Hndl.BtnSaveAs) THEN
	IF (CSV_Hndl.ReqSaveAs = 1) THEN
		CSV_Hndl.ReqSaveAs := 0;
		NewRecipe;	//call action: show layer and alpha pad
	END_IF;
	IF ((CSV_Hndl.NewFileNameEntered = TRUE) OR (CSV_Hndl.StatusNewFileName = 16384)) THEN
		CSV_Hndl.LayerNewFileName := INVISIBLE;
		//Name entered or escaped function ?
		IF (CSV_Hndl.NewFileNameEntered = TRUE) THEN
			//write to file
			CSV_Hndl.ReqSaveRecipeAs := TRUE;
			CSV_Hndl.SetListBoxIdxToZero := TRUE;                                        ///  HIER !!!!!!
			CSV_Hndl.ValueChanged := FALSE;
		END_IF;

		CSV_Hndl.NewFileNameEntered := FALSE;
	END_IF;
END_IF;

//---------------------------------
//navigation throught listbox 1 (recipe files)
IF (CSV_Hndl.ScrollHomeLbo1 = 1) THEN
	CSV_Hndl.ScrollHomeLbo1 := 0;
	CSV_Hndl.ListboxIdx := 0;
END_IF;

IF (CSV_Hndl.ScrollUpLbo1 = 1) THEN
	CSV_Hndl.ScrollUpLbo1 := 0;
		IF (CSV_Hndl.ListboxIdx > 0) THEN
		CSV_Hndl.ListboxIdx := CSV_Hndl.ListboxIdx - 1;
	END_IF;
END_IF;

IF (CSV_Hndl.ScrollDownLbo1 = 1) THEN
	CSV_Hndl.ScrollDownLbo1 := 0;
	IF (CSV_Hndl.ListboxIdx < CSV_Hndl.ListboxMaxLines) THEN
		CSV_Hndl.ListboxIdx := CSV_Hndl.ListboxIdx + 1;
	END_IF;
END_IF;

IF (CSV_Hndl.ScrollEndLbo1 = 1) THEN
	CSV_Hndl.ScrollEndLbo1 := 0;
	CSV_Hndl.ListboxIdx := CSV_Hndl.ListboxMaxLines;
END_IF;

	//---------------------------------
	//navigation throught listbox 2 (sections in recipe structure)
	IF (CSV_Hndl.ScrollHomeLbo2 = 1) THEN
		ProgParaIndexSearchDirection	:= mcPOSITIVE_DIR;
		CSV_Hndl.ScrollHomeLbo2 := 0;
		CSV_Hndl.ListboxProgParaIdx := 0;
	END_IF;

	IF (CSV_Hndl.ScrollUpLbo2 = 1) THEN
		ProgParaIndexSearchDirection	:= mcNEGATIVE_DIR;
		CSV_Hndl.ScrollUpLbo2 := 0;
			IF (CSV_Hndl.ListboxProgParaIdx > 0) THEN
			CSV_Hndl.ListboxProgParaIdx := CSV_Hndl.ListboxProgParaIdx - 1;
		END_IF;
	END_IF;

	IF (CSV_Hndl.ScrollDownLbo2 = 1) THEN
		ProgParaIndexSearchDirection	:= mcPOSITIVE_DIR;
		CSV_Hndl.ScrollDownLbo2 := 0;
		IF (CSV_Hndl.ListboxProgParaIdx  < CSV_Hndl.ListboxProgParaMaxLines) THEN
			CSV_Hndl.ListboxProgParaIdx  := CSV_Hndl.ListboxProgParaIdx  + 1;
		END_IF;
	END_IF;

	IF (CSV_Hndl.ScrollEndLbo2 = 1) THEN
		ProgParaIndexSearchDirection	:= mcNEGATIVE_DIR;
		CSV_Hndl.ScrollEndLbo2 := 0;
		CSV_Hndl.ListboxProgParaIdx := CSV_Hndl.ListboxProgParaMaxLines;
	END_IF;

	//check if the text at the current listbox index exists
	SPR_CheckTextIndexValid_0.Enable	:= TRUE;
	SPR_CheckTextIndexValid_0.TG_id		:= TXT_GRP_PROGPARASECTIONS;
	SPR_CheckTextIndexValid_0.TGT_id	:= CSV_Hndl.ListboxProgParaIdx;
	SPR_CheckTextIndexValid_0.VCHandle	:= VCHandle;
	SPR_CheckTextIndexValid_0();

	IF ( (SPR_CheckTextIndexValid_0.Status <> vaERR_BUSY) AND NOT SPR_CheckTextIndexValid_0.Valid) THEN
		IF (ProgParaIndexSearchDirection = mcPOSITIVE_DIR) THEN
			IF (CSV_Hndl.ListboxProgParaIdx  < CSV_Hndl.ListboxProgParaMaxLines) THEN
				CSV_Hndl.ListboxProgParaIdx		:= CSV_Hndl.ListboxProgParaIdx + 1;
			ELSE
				CSV_Hndl.ListboxProgParaIdx		:= CSV_Hndl.ListboxProgParaIdx - 1;
				ProgParaIndexSearchDirection	:= mcNEGATIVE_DIR;
			END_IF;
		ELSE
			IF (CSV_Hndl.ListboxProgParaIdx > 0) THEN
				CSV_Hndl.ListboxProgParaIdx		:= CSV_Hndl.ListboxProgParaIdx - 1;
			ELSE
				CSV_Hndl.ListboxProgParaIdx		:= CSV_Hndl.ListboxProgParaIdx + 1;
				ProgParaIndexSearchDirection	:= mcPOSITIVE_DIR;
			END_IF;
		END_IF;
	END_IF;

FOR ii := 0 TO 20 DO
	CSV_Hndl.LayersProgPara[ii] := INVISIBLE;
END_FOR;
CSV_Hndl.LayersProgPara[CSV_Hndl.ListboxProgParaIdx] := VISIBLE;

//---------------------------------
//copy all recipes from CF to USB Stick
//-> task save2USB

//---------------------------------
//CSV_Hndl.StatusBmpTensionOnOff := BOOL_TO_UINT(NOT(RecipeEdit.dancer.cylinderTension));
//CSV_Hndl.StatusBmpRadiusCtrlOnOff := BOOL_TO_UINT(NOT(RecipeEdit.dancer.radiusCtrlOn));
//CSV_Hndl.StatusBmpReverseGrid1 := BOOL_TO_UINT(NOT(RecipeEdit.grid1.reverse));
//CSV_Hndl.StatusBmpReverseGrid2 := BOOL_TO_UINT(NOT(RecipeEdit.grid2.reverse));
//CSV_Hndl.StatusBmpReverseSpender1 := BOOL_TO_UINT(NOT(RecipeEdit.spender1.reverse));
//CSV_Hndl.StatusBmpReverseSpender2 := BOOL_TO_UINT(NOT(RecipeEdit.spender2.reverse));

END_PROGRAM
```

#### csv_hdl.typ - Local data types
```iecst
(********************************************************************
 * COPYRIGHT -- Bernecker + Rainer
 ********************************************************************
 * Program: csv_hdl
 * File: csv_hdl.typ
 * Author: beutert
 * Created: August 28, 2012
 ********************************************************************
 * Local data types of program csv_hdl
 ********************************************************************)

TYPE
	Link_typ : 	STRUCT
		Prev : USINT;
		Next : USINT;
	END_STRUCT;
END_TYPE
```

#### csv_hdl.var - Local variables
```iecst
(********************************************************************
 * COPYRIGHT -- Bernecker + Rainer
 ********************************************************************
 * Program: csv_hdl
 * File: csv_hdl.var
 * Author: beutert
 * Created: August 28, 2012
 ********************************************************************
 * Local variables of program csv_hdl
 ********************************************************************)
VAR
	ProgParaIndexSearchDirection : USINT;
	VCHandle : UDINT;
END_VAR
VAR CONSTANT
	TXT_GRP_PROGPARASECTIONS : UDINT := 13;
END_VAR
VAR
	DirCreate_0 : DirCreate;
	CSV_Header : CSV_Header_typ;
	CSV_Hndl : CSVHndl_typ;
	CSV_InitVariable : CSV_Init;
	CSV_ListCSVFile : CSV_ListFile;
	CSV_ReadCSVFile : CSV_ReadFile;
	CSV_SearchData : CSV_Search;
	CSV_SearchFile : SearchFileName;
	CSV_WriteCSVFile : CSV_WriteFile;
	CSVCheckFileVersion : CSV_CheckFile;
	CSVInitCheckFileVersion : CSV_InitCheckFile;
	DevLink_0 : DevLink;
	DevUnlink_0 : DevUnlink;
	Dyn_Usint : REFERENCE TO USINT;
	Error : UINT;
	FileDelete_0 : FileDelete;
	FileNameOld : STRING[80];
	FileNamesRead : ARRAY[0..99] OF STRING[46];
	i : INT;
	ii : USINT;
END_VAR
VAR CONSTANT
	INVISIBLE : USINT := 1;
END_VAR
VAR
	OldListBoxIdx : UINT;
	pNames : ARRAY[0..4] OF UDINT;
	SaveUserData : USINT;
	Sort_0 : Sort;
END_VAR
VAR CONSTANT
	ST_ASK_FOR_DELETE_FILE : UINT := 7;
	ST_ASK_FOR_OVERWRITE_FILE : UINT := 11;
	ST_CHECK_VERSION : UINT := 6;
	ST_COMMAND : UINT := 0;
	ST_DELETE_FILE : UINT := 8;
	ST_ERROR : UINT := 255;
	ST_LINK_DEVICE : UINT := 16;
	ST_LIST_FILE : UINT := 1;
	ST_LIST_FILE_SORT : UINT := 2;
	ST_READ_FILE : UINT := 5;
	ST_REPLACE_WRONG_CHARS : UINT := 13;
	ST_SEARCH_DATA : UINT := 3;
	ST_SEARCH_FILE_ON_USB : UINT := 12;
	ST_SORT_FILE_NAMES : UINT := 9;
	ST_UNLINK_DEVICE : UINT := 15;
	ST_WRITE_FILE : UINT := 4;
END_VAR
VAR
	Step : UINT;
	StepOld : UINT;
	StructSizes : ARRAY[0..4] OF UDINT;
	szDevLinkPara : STRING[80];
	szFileDevice : STRING[80];
	tmpChar : STRING[1];
	tmpRecipe : rcp_prog_typ := (0);
	tmpRecipeOld : rcp_prog_typ := (0);
	tmpString : STRING[50];
END_VAR
VAR CONSTANT
	VISIBLE : USINT := 0;
END_VAR
VAR
	xSorted : BOOL;
	Layer_Password : BOOL;
	HWString : STRING[20];
	HWInfo_0 : HWInfo;
	InputPassword : STRING[8];
	Show_Layer_password : INT;
	Level_Passwort : INT := 10;
	SPR_CheckTextIndexValid_0 : SPR_CheckTextIndexValid;
END_VAR
```

#### NewRecipe.st
```iecst
(********************************************************************
 * COPYRIGHT -- Bernecker + Rainer
 ********************************************************************
 * Program: csv_hndl
 * File: NewRecipe.st
 * Author: beutert
 * Created: August 21, 2012
 ********************************************************************
 * Implementation of program csv_hndl
 ********************************************************************)

 (* Add a new action to your IEC program or library *)
ACTION NewRecipe:
	CSV_Hndl.FileNameNew := '';
	CSV_Hndl.LayerNewFileName := VISIBLE;	//show layer
	CSV_Hndl.StatusNewFileName := CSV_Hndl.StatusNewFileName  OR 2#0000000000001000; //show alphapad
END_ACTION
```

#### DefRecipe.st
```iecst
(********************************************************************
 * COPYRIGHT -- Bernecker + Rainer
 ********************************************************************
 * Program: csv_hndl
 * File: DefRecipe.st
 * Author: beutert
 * Created: August 24, 2012
 ********************************************************************
 * Implementation of program csv_hndl
 *
 * History:
 * 2012-08-24 /beutert/
 *		Task created
 * 2012-11-01 /schoenefeldr/
 *		use actual settings instead of general default values
 ********************************************************************)

 (* sets default values to recipe struct *)
ACTION DefRecipe:

	// 2012-11-01 /schoenefeldr/
	// Copy values for default application recipe from actual settings
	memcpy(ADR(tmpRecipe), ADR(gApplRecipe), SIZEOF(tmpRecipe));

(*	memset(ADR(tmpRecipe), 0, SIZEOF(tmpRecipe));

	// 2012-09-18 /schoenefeldr/
	// Set default values for special input values
	tmpRecipe.general.maxVelocity			:= DEFAULT_MASTER_MAX_VELO;
	tmpRecipe.general.masterAcceleration 	:= DEFAULT_MASTER_AUTO_MODE_ACC;
	// Set default values for modes
	tmpRecipe.cutUnit1.mode		:= OPM_CUT_SYNC_CUT;
	tmpRecipe.cutUnit2.mode		:= OPM_CUT_SYNC_CUT;
	tmpRecipe.endModule.mode	:= OPM_END_MODULE_BELTS;
	tmpRecipe.grid1.mode		:= OPM_WIND_WINDER;
	tmpRecipe.grid2.mode		:= OPM_WIND_WINDER;
	tmpRecipe.longCut.mode		:= OPM_LONG_CUT_ENABLED;
	tmpRecipe.markpoint1.mode	:= OPM_RM_SENSOR_CONTROL;
	tmpRecipe.markpoint2.mode	:= OPM_RM_SENSOR_CONTROL;
	tmpRecipe.spender1.mode		:= OPM_WIND_BRAKE;
	tmpRecipe.spender2.mode		:= OPM_WIND_BRAKE;
	tmpRecipe.spender3.mode		:= OPM_WIND_BRAKE;
	tmpRecipe.tensionMeas.mode	:= OPM_WEB_TENSION_ENABLED;
*)

END_ACTION
```

### Program Logical/pkgRecipe/tool_hdl (IEC) - file handling

#### tool_hdl.st - Implementation code
```iecst
(********************************************************************
 * COPYRIGHT -- Bernecker + Rainer
 ********************************************************************
 * Program: TOOL_Hdl
 * File: TOOL_Hdl.st
 * Author: beutert
 * Created: August 28, 2012
 ********************************************************************
 * Implementation of program TOOL_Hdl
 ********************************************************************)

PROGRAM _INIT

	TOOL_Hndl.LayerMessageBoxOverwrite := INVISIBLE;
	TOOL_Hndl.LayerMessageBoxDeleteFile := INVISIBLE;
	TOOL_Hndl.LayerNewFileName := INVISIBLE;
	TOOL_Hndl.LayerMessageBoxSaveFile := INVISIBLE;

	HWInfo_0.enable := TRUE;
	HWInfo_0.first := TRUE;
	HWInfo_0.pName := ADR(HWString);
	HWInfo_0();

	DirCreate_0.pDevice	:= ADR('USERPART');
	DirCreate_0.pName	:= ADR('Tools');
	DirCreate_0.enable	:= TRUE;
	REPEAT
		DirCreate_0();
	UNTIL (DirCreate_0.status <> ERR_FUB_BUSY) END_REPEAT;

	strcpy(ADR(szFileDevice), ADR('DIR_TOOL'));
	IF HWString = 'AR000' THEN
		strcpy(ADR(szDevLinkPara), ADR('/DEVICE=C:\\temp\\Tools'));
	ELSE
		strcpy(ADR(szDevLinkPara), ADR('/DEVICE=F:\\Tools'));
	END_IF

	DevLink_0.enable 	:= 1;
	DevLink_0.pDevice := ADR(szFileDevice);
	DevLink_0.pParam 	:= ADR(szDevLinkPara);
	REPEAT
		DevLink_0();
	UNTIL (DevLink_0.status <> ERR_FUB_BUSY) END_REPEAT;

	strcpy(ADR(CSV_Header.CustomerName),ADR('Spilker'));
	strcpy(ADR(CSV_Header.MachineNumber),ADR('Herpa Print'));
	strcpy(ADR(CSV_Header.SW_Version),ADR('Version V1.00'));

	//strcpy(ADR(RecipeEdit.MachineString),ADR('machine1'));

	pNames[0] :=  ADR('tool_hdl:tmpTool');		//Name der zu sichernden PV
//	pNames[1] :=  ADR('CSV_SearchData');				//mehrere möglich

	StructSizes[0] := SIZEOF(tmpTool);				//Größe der zu sichernden PV
//	StructSizes[1] := SIZEOF(CSV_SearchData);

	CSV_InitVariable.pStructName := ADR(pNames);
	CSV_InitVariable.NumOfStructs := 1;					//Anzahl der zu sichernden Elemente, wenn CSV_SearchData auch gesichert werden soll, muss hier 2 stehen
	CSV_InitVariable.FullNameLenght := 0;
	CSV_InitVariable.Options := 0;
	CSV_InitVariable();

  IF (CSV_InitVariable.status > 0) AND (CSV_InitVariable.status < ERR_FUB_BUSY) THEN
  	Step := ST_ERROR;
  ELSE
   	Step := ST_COMMAND;
	END_IF;

//Speicherplatz allokieren
	CSVInitCheckFileVersion.enable := 1;
	CSVInitCheckFileVersion.MemCounter := CSV_InitVariable.MemCounter;
	CSVInitCheckFileVersion();

  IF (CSVInitCheckFileVersion.status < 65535) AND (CSVInitCheckFileVersion.status > 0) THEN
    Step := ST_ERROR;
  ELSE
   	Step := ST_COMMAND;
		CSVInitCheckFileVersion.enable := 1;
		CSVInitCheckFileVersion.MemCounter := CSV_InitVariable.MemCounter;
		CSVInitCheckFileVersion();
	END_IF;

  IF (CSVInitCheckFileVersion.status < ERR_FUB_BUSY) AND (CSVInitCheckFileVersion.status > 0) THEN
    Step := ST_ERROR;
  ELSE
    Step := ST_COMMAND;
		TOOL_Hndl.ReqDirRead := TRUE;
		xSorted := TRUE;
		OldListBoxIdx := 16#FFFF;
	END_IF;

END_PROGRAM

PROGRAM _CYCLIC

CASE Step OF

	(****************************************/
	/* command interface                    */
	/****************************************)
	ST_COMMAND:	(*0*)
		IF (TOOL_Hndl.ReqDirRead) THEN
			IF (xSorted = TRUE) THEN
				Step := ST_LIST_FILE_SORT;
			ELSE
				Step := ST_LIST_FILE;
			END_IF;

		ELSIF (TOOL_Hndl.ReqDelRecipe) THEN
			TOOL_Hndl.ReqDelRecipe := FALSE;
			strcpy(ADR(TOOL_Hndl.FileNameDelete),ADR(TOOL_Hndl.ListboxFileNames[TOOL_Hndl.ListboxIdx]));
			strcat(ADR(TOOL_Hndl.FileNameDelete),ADR('.csv'));
			TOOL_Hndl.LayerMessageBoxDeleteFile := VISIBLE;	//Message einblenden
		  TOOL_Hndl.FileDelete := 0;
			Step := ST_ASK_FOR_DELETE_FILE;

		ELSIF (TOOL_Hndl.ReqCreateNew) THEN
			TOOL_Hndl.ReqCreateNew := FALSE;
//			memcpy(ADR(tmpTool), ADR(RecipeNew), SIZEOF(tmpTool));	//copy data structure
			Step := ST_SEARCH_DATA;

		ELSIF (TOOL_Hndl.ReqParaWrite) THEN
			memcpy(ADR(tmpTool), ADR(ToolEdit), SIZEOF(tmpTool)); 	//copy data structure global to local
			strcpy(ADR(TOOL_Hndl.FileNameNew),ADR(TOOL_Hndl.ListboxFileNames[TOOL_Hndl.ListboxIdx]));
			strcat(ADR(TOOL_Hndl.FileNameNew),ADR('.csv'));
			TOOL_Hndl.OverwriteFile := TRUE;
			Step := ST_SEARCH_DATA;

		ELSIF (TOOL_Hndl.ReqParaWriteAfterValueChanged) THEN
			TOOL_Hndl.ReqParaWriteAfterValueChanged := FALSE;
			memcpy(ADR(tmpTool), ADR(tmpToolOld), SIZEOF(tmpTool)); 	//copy data structure
			strcpy(ADR(TOOL_Hndl.FileNameNew),ADR(FileNameOld));
			strcat(ADR(TOOL_Hndl.FileNameNew),ADR('.csv'));
			TOOL_Hndl.OverwriteFile := TRUE;
			Step := ST_SEARCH_DATA;

		ELSIF (TOOL_Hndl.ReqSaveRecipeAs) THEN
			TOOL_Hndl.ReqSaveRecipeAs := FALSE;
			memcpy(ADR(tmpTool), ADR(ToolEdit), SIZEOF(tmpTool));	//copy data structure
			Step := ST_SEARCH_DATA;

		ELSIF (TOOL_Hndl.ReqParaRead) THEN
			Step := ST_READ_FILE;

//		ELSIF(Start_CheckVersion)THEN
//			Step:= ST_CHECK_VERSION;
		END_IF;

	(****************************************/
	/* list all CSV-files in a array-string */
	/****************************************)

	(*OHNE SORTIERUNG:*)
	(*csv-Dateien auf Device auflisten*)
	ST_LIST_FILE:	(*1*)
		StepOld := Step;
   	CSV_ListCSVFile.pStringArray := ADR(TOOL_Hndl.ListboxFileNames[0]);
   	CSV_ListCSVFile.SizeStringArray := SIZEOF(TOOL_Hndl.ListboxFileNames);
   	CSV_ListCSVFile.ArrayNum := SIZEOF(TOOL_Hndl.ListboxFileNames) / SIZEOF(TOOL_Hndl.ListboxFileNames[0]);
   	CSV_ListCSVFile.NumListboxLines := 10;
		CSV_ListCSVFile.pFileDevice := ADR(szFileDevice);
   	CSV_ListCSVFile.MaxNameLenght := 28;
   	CSV_ListCSVFile.command := FiJOB_CREATE_FILE_LIST; //2
   	CSV_ListCSVFile();

		IF (CSV_ListCSVFile.CSV_FileNum > 0) THEN
	    TOOL_Hndl.ListboxMaxLines := CSV_ListCSVFile.CSV_FileNum  - 1;
	  ELSE
	  	TOOL_Hndl.ListboxMaxLines := 0;
	  END_IF;

		//no error
	  IF (CSV_ListCSVFile.status = 0) THEN
			TOOL_Hndl.ReqDirRead := 0;

			IF (TOOL_Hndl.SetListBoxIdxToZero) THEN
				TOOL_Hndl.SetListBoxIdxToZero := FALSE;
				TOOL_Hndl.ListboxIdx := 0;
//				TOOL_Hndl.ListboxProgParaIdx := 0;
				TOOL_Hndl.ReqParaRead := TRUE;
			END_IF;

	  	Step := ST_COMMAND;
		END_IF;

	   //error
	   IF ( (CSV_ListCSVFile.status <> 0) AND (CSV_ListCSVFile.status <> 65535) ) THEN
	      TOOL_Hndl.ReqDirRead := 0;
	      Step := ST_ERROR;
	   END_IF;

	(*MIT SORTIERUNG:*)
	(*csv-Dateien auf Device auflisten*)
	ST_LIST_FILE_SORT:	(*2*)
		StepOld := Step;
   	CSV_ListCSVFile.pStringArray := ADR(FileNamesRead);
   	CSV_ListCSVFile.SizeStringArray := SIZEOF(FileNamesRead);
   	CSV_ListCSVFile.ArrayNum := SIZEOF(FileNamesRead) / SIZEOF(FileNamesRead[0]);
   	CSV_ListCSVFile.NumListboxLines := 10;
		CSV_ListCSVFile.pFileDevice := ADR(szFileDevice);
   	CSV_ListCSVFile.MaxNameLenght := 28;
   	CSV_ListCSVFile.command := 2;
   	CSV_ListCSVFile();

		IF (CSV_ListCSVFile.CSV_FileNum > 0) THEN
	    TOOL_Hndl.ListboxMaxLines := CSV_ListCSVFile.CSV_FileNum  - 1;
	  ELSE
	  	TOOL_Hndl.ListboxMaxLines := 0;
	  END_IF;

	  //no error
	  IF (CSV_ListCSVFile.status = 0) THEN
  		Step := ST_SORT_FILE_NAMES;
		END_IF;

	   //error
	   IF ( (CSV_ListCSVFile.status <> 0) AND (CSV_ListCSVFile.status <> 65535) ) THEN
	      TOOL_Hndl.ReqDirRead := 0;
	      Step := ST_ERROR;
	   END_IF;

	(****************************************/
	/* sort FileNames                    */
	/****************************************)
	ST_SORT_FILE_NAMES:	(*9*)
		StepOld := Step;
    Sort_0.enable := TRUE;
		Sort_0.pStringArray := ADR(FileNamesRead);
		Sort_0.StringLen := SIZEOF(FileNamesRead[0]);
		Sort_0.ArrayLen := SIZEOF(FileNamesRead);
		Sort_0();

	  IF (Sort_0.Status = 0) THEN
	  	TOOL_Hndl.ReqDirRead := 0;
			memcpy(ADR(TOOL_Hndl.ListboxFileNames), ADR(FileNamesRead), SIZEOF(FileNamesRead));

			IF (TOOL_Hndl.SetListBoxIdxToZero) THEN
				TOOL_Hndl.SetListBoxIdxToZero := FALSE;
				TOOL_Hndl.ListboxIdx := 0;
//				TOOL_Hndl.ListboxProgParaIdx := 0;
				TOOL_Hndl.ReqParaRead := TRUE;
			END_IF;

	   	Step := ST_COMMAND;
	  END_IF;

	(*****************************************/
	/* search for the data from the variable */
	/*****************************************)
	ST_SEARCH_DATA:	(*3*)
		StepOld := Step;
//		memcpy(ADR(tmpTool), ADR(ToolEdit), SIZEOF(tmpTool)); globale Datenstruktur auf lokale umkopieren
   	CSV_SearchData.pStructName := CSV_InitVariable.pStructName;
   	CSV_SearchData.NumOfStructs := CSV_InitVariable.NumOfStructs;
   	CSV_SearchData.pStructMem := CSV_InitVariable.pStructMem;
   	CSV_SearchData.MemLen := CSV_InitVariable.MemCounter;
   	CSV_SearchData.FullNameLenght := 0;
   	CSV_SearchData.Separator := 59;	//';';
   	CSV_SearchData.Options := 0;
   	CSV_SearchData.FileHeader := HEADER;
   	CSV_SearchData.pMaschineNo := ADR(CSV_Header.CustomerName);
   	CSV_SearchData.pComment := ADR(CSV_Header.MachineNumber);
   	CSV_SearchData.pVersion := ADR(CSV_Header.SW_Version);
   	CSV_SearchData();

   	//no error
   	IF (CSV_SearchData.status = 0) THEN
			strcpy(ADR(TOOL_Hndl.FileNameSave), ADR(TOOL_Hndl.FileNameNew));
			TOOL_Hndl.ReqParaWrite := FALSE;
			Step := ST_REPLACE_WRONG_CHARS;
   	END_IF;

   	//error
	  IF ( (CSV_SearchData.status <> 0) AND (CSV_SearchData.status <> 65535) ) THEN
	  	Step := ST_ERROR;
		END_IF;

	(****************************************/
	/* Replace Wrong Signs                  */
	/****************************************)
	ST_REPLACE_WRONG_CHARS:	(*13*)
		StepOld := Step;
		IF (strlen(ADR(TOOL_Hndl.FileNameSave)) <> 0) THEN
			//control, if the filename has the right extension
			strcpy(ADR(tmpString), ADR(''));

			FOR i:=0 TO strlen(ADR(TOOL_Hndl.FileNameSave))-1 DO
				Dyn_Usint ACCESS (ADR(TOOL_Hndl.FileNameSave) + i);
				strcpy(ADR(tmpChar), ADR(''));
				memcpy(ADR(tmpChar), ADR(TOOL_Hndl.FileNameSave) + i, 1);
//				IF ( ((Dyn_Usint >= ADR('0') ) AND (Dyn_Usint <= ADR('9') )) OR
//				     ((Dyn_Usint >= ADR('A') ) AND (Dyn_Usint <= ADR('Z') )) OR
//						 ((Dyn_Usint >= ADR('a') ) AND (Dyn_Usint <= ADR('z') )) OR
//						 ( Dyn_Usint  = ADR('_') ) OR  (Dyn_Usint = ADR('-')   ) OR
//						 ( Dyn_Usint  = ADR('.') ) OR  (Dyn_Usint = 0) ) THEN
					IF (((Dyn_Usint >= 48) AND (Dyn_Usint <= 57)) OR
						  ((Dyn_Usint >= 65) AND (Dyn_Usint <= 90)) OR
						  ((Dyn_Usint >= 97) AND (Dyn_Usint <= 122)) OR
						   (Dyn_Usint  = 95) OR (Dyn_Usint = 45) OR
						   (Dyn_Usint  = 46) OR (Dyn_Usint = 0)) THEN
					//valid chars
					tmpString := CONCAT(tmpString, tmpChar);
				ELSE
					//non valid chars
					tmpString := CONCAT(tmpString, '-');
				END_IF;
			END_FOR;
		END_IF;	//(strlen(ADR(TOOL_Hndl.FileNameSave)) <> 0)

		Step := ST_SEARCH_FILE_ON_USB;
		strcpy (ADR(TOOL_Hndl.FileNameSave),ADR(tmpString));

	(****************************************/
	/* search filenames                    */
	/****************************************)
	ST_SEARCH_FILE_ON_USB:	(*12*)
		StepOld := Step;
	  CSV_SearchFile.pFileName := ADR(TOOL_Hndl.FileNameSave);
		CSV_SearchFile.pDevice := ADR(szFileDevice);
 		CSV_SearchFile();

	  //no error No file Found
	  IF (CSV_SearchFile.status = 0) THEN
	  	Step := ST_WRITE_FILE;
		END_IF;
	  //no error File Found
	  IF (CSV_SearchFile.status = 1) THEN
			IF (TOOL_Hndl.OverwriteFile) THEN
				TOOL_Hndl.OverwriteFile := FALSE;
				Step := ST_WRITE_FILE;
			ELSE
				TOOL_Hndl.LayerMessageBoxOverwrite := VISIBLE;	//Message einblenden
			  TOOL_Hndl.FileOverWrite := 0;
		  	Step := ST_ASK_FOR_OVERWRITE_FILE;
			END_IF;
		END_IF;
	  //error
	  IF ((CSV_SearchFile.status > 1) AND (CSV_SearchFile.status <> ERR_FUB_BUSY)) THEN
	  	Step := ST_ERROR;
	  END_IF;

	(****************************************/
	/* ask for overwrite file               */
	/****************************************)
	ST_ASK_FOR_OVERWRITE_FILE:	(*11*)
		StepOld := Step;
		IF (TOOL_Hndl.LayerMessageBoxOverwrite = INVISIBLE) THEN
			IF (TOOL_Hndl.FileOverWrite = 0) THEN
				TOOL_Hndl.ReqNewRecipe := 1;	//start dialogue again
				Step := ST_COMMAND;
			ELSE
   			Step := ST_WRITE_FILE;
				TOOL_Hndl.FileOverWrite := 0;
	    END_IF;
		END_IF;

	(*****************************************/
	/* write the searched data in a CSV-file */
	/*****************************************)
	ST_WRITE_FILE:	(*4*)
		StepOld := Step;
	 	CSV_WriteCSVFile.pFileName := ADR(TOOL_Hndl.FileNameSave);
	  CSV_WriteCSVFile.pDevice := ADR(szFileDevice);
	 	CSV_WriteCSVFile.pStructMem := CSV_InitVariable.pStructMem;
	 	CSV_WriteCSVFile.MemLen := CSV_SearchData.FileLen;
	 	CSV_WriteCSVFile.Mode := FILE_OW;
	 	CSV_WriteCSVFile();

	  //no error
	  IF (CSV_WriteCSVFile.status = 0) THEN
	  	TOOL_Hndl.ReqParaWrite := FALSE;
			TOOL_Hndl.ReqDirRead := TRUE;		//read directory again after writing a (new) file
	    Step := ST_COMMAND;
	  END_IF;
	  //error
	  IF ((CSV_WriteCSVFile.status <> 0) AND (CSV_WriteCSVFile.status <> 65535)) THEN
			TOOL_Hndl.ReqParaWrite := FALSE;
    	//Es sind nur Zeichen und Zahlen erlaubt
			IF (CSV_WriteCSVFile.status = 5004) THEN
				Step :=  ST_ERROR;
			END_IF;
			Step := ST_ERROR;
	 	END_IF;

	(*****************************************/
	/* read a CSV-file                       */
	/*****************************************)
	ST_READ_FILE:	(*5*)
		StepOld := Step;
	  CSV_ReadCSVFile.pFileName := ADR(TOOL_Hndl.ListboxFileNames[TOOL_Hndl.ListboxIdx]);
   	CSV_ReadCSVFile.pDevice := ADR(szFileDevice);
   	CSV_ReadCSVFile.No_DatatypControl := 1;
//   	CSV_ReadCSVFile.Options := 0;
   	CSV_ReadCSVFile.IgnoreError := 1;
   	CSV_ReadCSVFile.Separator := 59;	//';';
   	CSV_ReadCSVFile();

   	//no error
   	IF (CSV_ReadCSVFile.status = 0) THEN
     	TOOL_Hndl.ReqParaRead := 0;
			memcpy(ADR(ToolEdit), ADR(tmpTool), SIZEOF(ToolEdit));
			SaveUserData := 1;
      Step := ST_COMMAND;
   	END_IF;

   	//error
   	IF ((CSV_ReadCSVFile.status <> 0) AND (CSV_ReadCSVFile.status <> 65535)) THEN
      TOOL_Hndl.ReqParaRead := 0;
      Step := ST_ERROR;
	 END_IF;

	(*****************************************/
	/* read a CSV-file                       */
	/*****************************************)
	ST_CHECK_VERSION:	(*6*)
		StepOld := Step;
		CSVCheckFileVersion.enable := 1;
		CSVCheckFileVersion.pFileName := ADR('csv1.CSV');
		CSVCheckFileVersion.pDevice := ADR(szFileDevice);
		CSVCheckFileVersion.pStructSizes := ADR(StructSizes);
		CSVCheckFileVersion.NumOfStruct := CSV_InitVariable.NumOfStructs;
		CSVCheckFileVersion.pVersion := ADR('V0.02.2');
		CSVCheckFileVersion.pFileBuffer := CSVInitCheckFileVersion.pFileBuffer;
		CSVCheckFileVersion.FileBufferSize := CSVInitCheckFileVersion.FileBufferSize;
		CSVCheckFileVersion();

	  //no error
	 	IF (CSVCheckFileVersion.status = 0) THEN
	   	Step := ST_COMMAND;
	 	END_IF;

	  //error
	  IF ((CSVCheckFileVersion.status <> 0) AND (CSVCheckFileVersion.status <> 65535)) THEN
			Step := ST_ERROR;
   	END_IF;

	(****************************************/
	/* ask for delete file                  */
	/****************************************)
	ST_ASK_FOR_DELETE_FILE:	(*7*)
		StepOld := Step;
		IF (TOOL_Hndl.LayerMessageBoxDeleteFile = INVISIBLE) THEN
			IF (TOOL_Hndl.FileDelete = 0) THEN
				Step := ST_COMMAND;
			ELSE
				TOOL_Hndl.FileDelete := 0;
   			Step := ST_DELETE_FILE;
	    END_IF;
		END_IF;

	(*****************************************/
	/* delete a CSV-file                       */
	/*****************************************)
	ST_DELETE_FILE:	(*8*)
		StepOld := Step;
		FileDelete_0.enable 	:= 1;
		FileDelete_0.pDevice 	:= ADR(szFileDevice);
		FileDelete_0.pName 		:= ADR(TOOL_Hndl.FileNameDelete);
		FileDelete_0();

	  //no error
	 	IF (FileDelete_0.status = 0) THEN
			TOOL_Hndl.ReqDirRead := TRUE;		//read directory again after deleting a file
			TOOL_Hndl.SetListBoxIdxToZero := TRUE;
	   	Step := ST_COMMAND;
	 	END_IF;

	  //error
	  IF ((FileDelete_0.status <> 0) AND (FileDelete_0.status <> ERR_FUB_BUSY)) THEN
			Step := ST_ERROR;
   	END_IF;

	(****************************************/
	/* change the file device               */
	/****************************************)
	ST_UNLINK_DEVICE:	(*15*)
		StepOld := Step;
		DevUnlink_0.enable := 1;
		DevUnlink_0.handle := DevLink_0.handle;
		DevUnlink_0();

	  //no error
		IF (DevUnlink_0.status = 0) THEN
			Step := ST_LINK_DEVICE;
		ELSIF (DevUnlink_0.status = ERR_FUB_BUSY) THEN
			//
		ELSE
			Step := ST_ERROR;
		END_IF;

	ST_LINK_DEVICE:	(*16*)
		StepOld := Step;
		DevLink_0.enable 	:= 1;
		DevLink_0.pDevice := ADR(szFileDevice);
		DevLink_0.pParam 	:= ADR(szDevLinkPara);
		DevLink_0();

	  //no error
		IF (DevLink_0.status = 0) THEN
			TOOL_Hndl.SetListBoxIdxToZero := TRUE;
			TOOL_Hndl.ReqDirRead := TRUE;
			Step := ST_COMMAND;
		ELSIF (DevLink_0.status = ERR_FUB_BUSY) THEN
			//
		ELSE
			Step := ST_ERROR;
		END_IF;

	(****************************************/
	/* error counter                        */
	/****************************************)
	ST_ERROR:	(*255*)
	   Error := Error + 1;
	   Step := ST_COMMAND;

END_CASE;

(*************************************************************************
 ************************************************************************)
//copy the name of the selected csv file into a variable
IF ((TOOL_Hndl.ListboxIdx >= 0) AND (TOOL_Hndl.ListboxIdx < 100)) THEN
	strcpy(ADR(TOOL_Hndl.FileNameSelected), ADR(TOOL_Hndl.ListboxFileNames[TOOL_Hndl.ListboxIdx]));
ELSE
	strcpy(ADR(TOOL_Hndl.FileNameSelected),ADR('index out of range'));
END_IF;

//another recipe was selected in the list
IF (OldListBoxIdx <> TOOL_Hndl.ListboxIdx) THEN
	IF (TOOL_Hndl.ValueChanged) THEN			//a value was changed
		TOOL_Hndl.ValueChanged := FALSE;
		memcpy(ADR(tmpToolOld), ADR(ToolEdit), SIZEOF(tmpToolOld)); 	//copy data structure global to local
		strcpy(ADR(FileNameOld),  ADR(TOOL_Hndl.ListboxFileNames[OldListBoxIdx]));
		TOOL_Hndl.LayerMessageBoxSaveFile := VISIBLE;	//show messagebox
	END_IF;
	IF (TOOL_Hndl.LayerMessageBoxSaveFile = INVISIBLE) THEN
		OldListBoxIdx := TOOL_Hndl.ListboxIdx;
		TOOL_Hndl.ReqParaRead := TRUE;

//		TOOL_Hndl.ListboxProgParaIdx := 0;	//set index of second listbox to 0
	END_IF;
END_IF;

//---------------------------------
//create a new recipe
IF(TOOL_Hndl.BtnNew) THEN
	IF (TOOL_Hndl.ReqNewRecipe = 1) THEN
		TOOL_Hndl.ReqNewRecipe := 0;
		NewTool;	//call action: show layer and alpha pad
	END_IF;
	IF ((TOOL_Hndl.NewFileNameEntered = TRUE) OR (TOOL_Hndl.StatusNewFileName = 16384)) THEN
		TOOL_Hndl.LayerNewFileName := INVISIBLE;
		//Name entered or escaped function ?
		IF (TOOL_Hndl.NewFileNameEntered = TRUE) THEN
			//create structure with default values and write to file
			DefTool;
			TOOL_Hndl.ReqCreateNew := TRUE;
			TOOL_Hndl.SetListBoxIdxToZero := TRUE;
		END_IF;

		TOOL_Hndl.NewFileNameEntered := FALSE;
	END_IF;
END_IF;

//---------------------------------
//save a recipe under a new name
IF (TOOL_Hndl.BtnSaveAs) THEN
	IF (TOOL_Hndl.ReqSaveAs = 1) THEN
		TOOL_Hndl.ReqSaveAs := 0;
		NewTool;	//call action: show layer and alpha pad
	END_IF;
	IF ((TOOL_Hndl.NewFileNameEntered = TRUE) OR (TOOL_Hndl.StatusNewFileName = 16384)) THEN
		TOOL_Hndl.LayerNewFileName := INVISIBLE;
		//Name entered or escaped function ?
		IF (TOOL_Hndl.NewFileNameEntered = TRUE) THEN
			//write to file
			TOOL_Hndl.ReqSaveRecipeAs := TRUE;
			TOOL_Hndl.SetListBoxIdxToZero := TRUE;
			TOOL_Hndl.ValueChanged := FALSE;
		END_IF;

		TOOL_Hndl.NewFileNameEntered := FALSE;
	END_IF;
END_IF;

	//---------------------------------
	//navigation throught listbox 1 (tool files)
	IF (TOOL_Hndl.ScrollHomeLbo1 = 1) THEN
		TOOL_Hndl.ScrollHomeLbo1 := 0;
		TOOL_Hndl.ListboxIdx := 0;
	END_IF;

	IF (TOOL_Hndl.ScrollUpLbo1 = 1) THEN
		TOOL_Hndl.ScrollUpLbo1 := 0;
			IF (TOOL_Hndl.ListboxIdx > 0) THEN
			TOOL_Hndl.ListboxIdx := TOOL_Hndl.ListboxIdx - 1;
		END_IF;
	END_IF;

	IF (TOOL_Hndl.ScrollDownLbo1 = 1) THEN
		TOOL_Hndl.ScrollDownLbo1 := 0;
		IF (TOOL_Hndl.ListboxIdx < TOOL_Hndl.ListboxMaxLines) THEN
			TOOL_Hndl.ListboxIdx := TOOL_Hndl.ListboxIdx + 1;
		END_IF;
	END_IF;

	IF (TOOL_Hndl.ScrollEndLbo1 = 1) THEN
		TOOL_Hndl.ScrollEndLbo1 := 0;
		TOOL_Hndl.ListboxIdx := TOOL_Hndl.ListboxMaxLines;
	END_IF;

//---------------------------------
////navigation throught listbox 2 (sections in recipe structure)
//IF (TOOL_Hndl.ScrollHomeLbo2 = 1) THEN
//	TOOL_Hndl.ScrollHomeLbo2 := 0;
//	TOOL_Hndl.ListboxProgParaIdx := 0;
//END_IF;
//
//IF (TOOL_Hndl.ScrollUpLbo2 = 1) THEN
//	TOOL_Hndl.ScrollUpLbo2 := 0;
//		IF (TOOL_Hndl.ListboxProgParaIdx > 0) THEN
//		TOOL_Hndl.ListboxProgParaIdx := TOOL_Hndl.ListboxProgParaIdx - 1;
//	END_IF;
//END_IF;
//
//IF (TOOL_Hndl.ScrollDownLbo2 = 1) THEN
//	TOOL_Hndl.ScrollDownLbo2 := 0;
//	IF (TOOL_Hndl.ListboxProgParaIdx  < TOOL_Hndl.ListboxProgParaMaxLines) THEN
//		TOOL_Hndl.ListboxProgParaIdx  := TOOL_Hndl.ListboxProgParaIdx  + 1;
//	END_IF;
//END_IF;
//
//IF (TOOL_Hndl.ScrollEndLbo2 = 1) THEN
//	TOOL_Hndl.ScrollEndLbo2 := 0;
//	TOOL_Hndl.ListboxProgParaIdx := TOOL_Hndl.ListboxProgParaMaxLines;
//END_IF;

//FOR ii := 0 TO 20 DO
//	TOOL_Hndl.LayersProgPara[ii] := INVISIBLE;
//END_FOR;
//TOOL_Hndl.LayersProgPara[TOOL_Hndl.ListboxProgParaIdx] := VISIBLE;

//---------------------------------
//copy all tools from CF to USB Stick
//-> task save2USB

//---------------------------------
//TOOL_Hndl.StatusBmp := BOOL_TO_UINT(NOT(ToolEdit.toolingLayout));

END_PROGRAM
```

#### tool_hdl.var - Local variables
```iecst
(********************************************************************
 * COPYRIGHT -- Bernecker + Rainer
 ********************************************************************
 * Program: csv_hdl
 * File: csv_hdl.var
 * Author: beutert
 * Created: August 28, 2012
 ********************************************************************
 * Local variables of program csv_hdl
 ********************************************************************)
VAR
	DirCreate_0 : DirCreate;
	CSV_Header : CSV_Header_typ;
	CSV_InitVariable : CSV_Init;
	CSV_ListCSVFile : CSV_ListFile;
	CSV_ReadCSVFile : CSV_ReadFile;
	CSV_SearchData : CSV_Search;
	CSV_SearchFile : SearchFileName;
	CSV_WriteCSVFile : CSV_WriteFile;
	CSVCheckFileVersion : CSV_CheckFile;
	CSVInitCheckFileVersion : CSV_InitCheckFile;
	DevLink_0 : DevLink;
	DevUnlink_0 : DevUnlink;
	Dyn_Usint : REFERENCE TO USINT;
	Error : UINT;
	FileDelete_0 : FileDelete;
	FileNameOld : STRING[80];
	FileNamesRead : ARRAY[0..99] OF STRING[46];
	i : INT;
END_VAR
VAR CONSTANT
	INVISIBLE : USINT := 1;
END_VAR
VAR
	OldListBoxIdx : UINT;
	pNames : ARRAY[0..4] OF UDINT;
	SaveUserData : USINT;
	Sort_0 : Sort;
END_VAR
VAR CONSTANT
	ST_ASK_FOR_DELETE_FILE : UINT := 7;
	ST_ASK_FOR_OVERWRITE_FILE : UINT := 11;
	ST_CHECK_VERSION : UINT := 6;
	ST_COMMAND : UINT := 0;
	ST_DELETE_FILE : UINT := 8;
	ST_ERROR : UINT := 255;
	ST_LINK_DEVICE : UINT := 16;
	ST_LIST_FILE : UINT := 1;
	ST_LIST_FILE_SORT : UINT := 2;
	ST_READ_FILE : UINT := 5;
	ST_REPLACE_WRONG_CHARS : UINT := 13;
	ST_SEARCH_DATA : UINT := 3;
	ST_SEARCH_FILE_ON_USB : UINT := 12;
	ST_SORT_FILE_NAMES : UINT := 9;
	ST_UNLINK_DEVICE : UINT := 15;
	ST_WRITE_FILE : UINT := 4;
END_VAR
VAR
	Step : UINT;
	StepOld : UINT;
	StructSizes : ARRAY[0..4] OF UDINT;
	szDevLinkPara : STRING[80];
	szFileDevice : STRING[80];
	tmpChar : STRING[1];
	tmpTool : rcp_tool_typ := (0);
	tmpToolOld : rcp_tool_typ := (0);
	tmpString : STRING[50];
END_VAR
VAR CONSTANT
	VISIBLE : USINT := 0;
END_VAR
VAR
	xSorted : BOOL;
	TOOL_Hndl : TOOL_Hndl_typ;
	HWInfo_0 : HWInfo;
	HWString : STRING[20];
END_VAR
```

#### NewTool.st
```iecst
(********************************************************************
 * COPYRIGHT -- Bernecker + Rainer
 ********************************************************************
 * Program: tool_Hdl
 * File: NewTool.st
 * Author: beutert
 * Created: August 21, 2012
 ********************************************************************
 * Implementation of program tool_Hdl
 ********************************************************************)

 (* Add a new action to your IEC program or library *)
ACTION NewTool:
	TOOL_Hndl.FileNameNew := '';
	TOOL_Hndl.LayerNewFileName := VISIBLE;	//show layer
	TOOL_Hndl.StatusNewFileName := TOOL_Hndl.StatusNewFileName  OR 2#0000000000001000; //show alphapad
END_ACTION
```

#### DefTool.st
```iecst
(********************************************************************
 * COPYRIGHT -- Bernecker + Rainer
 ********************************************************************
 * Program: tool_hndl
 * File: DefTool.st
 * Author: beutert
 * Created: August 24, 2012
 ********************************************************************
 * Implementation of program tool_hndl
 ********************************************************************)

 (* sets default values to tool struct *)
ACTION DefTool:
	memset(ADR(tmpTool), 0, SIZEOF(tmpTool));

	// 2012-09-19 /schoenefeldr/
	// Default values for some parameters
	tmpTool.cogCutting			:= DEFAULT_COG_CUTTING;
	tmpTool.cogSupportSpindle	:= DEFAULT_COG_SUPP_SPINDLE;
	tmpTool.numberToolSegments	:= DEFAULT_COG_TOOL_SEGMENTS;

END_ACTION
```

### Program Logical/pkgRecipe/al_hdl (IEC) - alarm handling

#### al_hdl.st - Implementation code
```iecst
(********************************************************************
 * COPYRIGHT -- Bernecker + Rainer
 ********************************************************************
 * Program: al_hndl
 * File: al_hndl.st
 * Author: beutert
 * Created: August 28, 2012
 ********************************************************************
 * Implementation of program al_hndl
 *
 * History:
 * 2012-08-28 /beutert/
 *		Task created
 * 2012-10-30 /schoenefeldr/
 *		Use global diameter status variable for alarms
 ********************************************************************)

PROGRAM _INIT

AlarmBit_a[0] := AlarmBit_a[0];
QuitBit_a[0] := QuitBit_a[0];
WarningBit_a[0] := WarningBit_a[0];

END_PROGRAM

PROGRAM _CYCLIC

	// Erzeugung von Alarme,
	// Fehler 0
	IF FALSE THEN
	AlarmBit_a[0] := 1;
	END_IF;
	// Fehler 1
	IF FALSE THEN
		AlarmBit_a[1] := 1;
	END_IF;
	// Fehler 2
	IF FALSE THEN
		AlarmBit_a[2] := 1;
	END_IF;
	// Fehler 3
	IF FALSE THEN
		AlarmBit_a[3] := 1;
	END_IF;
	// Fehler 4
	IF FALSE THEN
		AlarmBit_a[4] := 1;
	END_IF;
	// Fehler 5
	IF FALSE THEN
		AlarmBit_a[5] := 1;
	END_IF;

	// Erzeugung von Warnungen,
	// Warnung 0
	IF FALSE THEN
		WarningBit_a[0] := 1;
	END_IF;

	// Warnung 1 UnWinder
	IF gMachine.Status.Diam.MainUnwind < gMachRecipe.mainUnwind.WarnDiam  THEN
		WarningBit_a[1] := 1;
	END_IF;
	// Warnung 2 Spender 1
//	IF gMachine.Status.Diam.Spend1 > gMachRecipe.spender1.WarnDiam  AND  (gApplRecipe.spender1.mode = 1) THEN
//		WarningBit_a[2] := 1;
//	END_IF;
	// Warnung 3 Gridwinder 1
	IF gMachine.Status.Diam.Grid1 > gMachRecipe.grid1.WarnDiam AND  (gApplRecipe.grid1.mode = OPM_WIND_WINDER) THEN
		WarningBit_a[3] := 1;
	END_IF;
	// Warnung 4 Spender 2
//	IF gMachine.Status.Diam.Spend2 > gMachRecipe.spender2.WarnDiam  AND  (gApplRecipe.spender2.mode = OPM_WIND_WINDER) THEN
//		WarningBit_a[4] := 1;
//	END_IF;
	// Warnung 5 Gridwinder 2
	IF gMachine.Status.Diam.Grid2 > gMachRecipe.grid2.StopDiam  AND  (gApplRecipe.grid2.mode = OPM_WIND_WINDER) THEN
		WarningBit_a[5] := 1;
	END_IF;

		// Warnung 6 Spender 3
//		IF gMachine.Status.Diam.Spend3 > gMachRecipe.spender3.WarnDiam  AND  (gApplRecipe.spender3.mode= OPM_WIND_WINDER) THEN
//			WarningBit_a[6] := 1;
//		END_IF;

		// Warnung 7 Top Winder 2
//			IF gMachine.Status.Diam.TUnwindTop	 > gMachRecipe.topTandemWind.WarnDiam AND ((gApplRecipe.endModule.mode =OPM_END_MODULE_TANDEM_WINDER) OR (gApplRecipe.endModule.mode =OPM_END_MODULE_TOP_WINDER))  THEN
//			WarningBit_a[7] := 1;
//		END_IF;
//
		// Warnung 8 Button Winder 2
//		IF gMachine.Status.Diam.TUnwindBot	 > gMachRecipe.botTandemWind.WarnDiam AND  ((gApplRecipe.endModule.mode = OPM_END_MODULE_TANDEM_WINDER) OR (gApplRecipe.endModule.mode = OPM_END_MODULE_BOT_WINDER)) THEN
//			WarningBit_a[8] := 1;
//		END_IF;

		// Warnung 9
		IF FALSE THEN
			WarningBit_a[9] := 1;
		END_IF;

END_PROGRAM
```

#### al_hdl.var - Local variables
```iecst
(********************************************************************
 * COPYRIGHT -- Bernecker + Rainer
 ********************************************************************
 * Program: al_hndl
 * File: al_hndl.var
 * Author: beutert
 * Created: August 28, 2012
 ********************************************************************
 * Local variables of program al_hndl
 ********************************************************************)
VAR CONSTANT
	MAX_ALARMS : UINT := 200;
	MAX_WARNINGS : UINT := 200;
END_VAR
VAR
	AlarmBit_a : ARRAY[0..MAX_ALARMS] OF BOOL;
	QuitBit_a : ARRAY[0..MAX_ALARMS] OF BOOL;
	WarningBit_a : ARRAY[0..MAX_WARNINGS] OF BOOL;
END_VAR
```

### Program Logical/pkgRecipe/picctrl (IEC, version 0.00.0)
